gfCNCPoint4[2434] = {X 524.9094, Y 36.3306, Z -5.5000, A 0.000, B 0.000, C 0.000 }
gfCNCPoint4[2435] = {X 523.9717, Y 36.0380, Z -5.5000, A 0.000, B 0.000, C 0.000 }
gfCNCPoint4[2436] = {X 523.1116, Y 35.5636, Z -5.5000, A 0.000, B 0.000, C 0.000 }
gfCNCPoint4[2437] = {X 522.3639, Y 34.9265, Z -5.5000, A 0.000, B 0.000, C 0.000 }
gfCNCPoint4[2438] = {X 521.7590, Y 34.1525, Z -5.5000, A 0.000, B 0.000, C 0.000 }
gfCNCPoint4[2439] = {X 521.3213, Y 33.2731, Z -5.5000, A 0.000, B 0.000, C 0.000 }
gfCNCPoint4[2440] = {X 521.0686, Y 32.3239, Z -5.5000, A 0.000, B 0.000, C 0.000 }
gfCNCPoint4[2441] = {X 521.0222, Y 31.9379, Z -5.5000, A 0.000, B 0.000, C 0.000 }
gfCNCPoint4[2442] = {X 521.0068, Y 31.5494, Z -5.5000, A 0.000, B 0.000, C 0.000 }
gfCNCPoint4[2443] = {X 521.0076, Y 24.4815, Z -5.5000, A 0.000, B 0.000, C 0.000 }
gfCNCPoint4[2444] = {X 521.0984, Y 23.6300, Z -5.5000, A 0.000, B 0.000, C 0.000 }
gfCNCPoint4[2445] = {X 521.3368, Y 22.8074, Z -5.5000, A 0.000, B 0.000, C 0.000 }
gfCNCPoint4[2446] = {X 521.7152, Y 22.0391, Z -5.5000, A 0.000, B 0.000, C 0.000 }
gfCNCPoint4[2447] = {X 521.1864, Y 22.1316, Z -5.5000, A 0.000, B 0.000, C 0.000 }
gfCNCPoint4[2448] = {X 520.6505, Y 22.1656, Z -5.5000, A 0.000, B 0.000, C 0.000 }
gfCNCPoint4[2449] = {X 519.9691, Y 22.1657, Z -5.5000, A 0.000, B 0.000, C 0.000 }
gfCNCPoint4[2450] = {X 519.5109, Y 22.1442, Z -5.5000, A 0.000, B 0.000, C 0.000 }
gfCNCPoint4[2451] = {X 519.0567, Y 22.0797, Z -5.5000, A 0.000, B 0.000, C 0.000 }
gfCNCPoint4[2452] = {X 518.1336, Y 21.8074, Z -5.5000, A 0.000, B 0.000, C 0.000 }
gfCNCPoint4[2453] = {X 517.2820, Y 21.3592, Z -5.5000, A 0.000, B 0.000, C 0.000 }
gfCNCPoint4[2454] = {X 516.5348, Y 20.7527, Z -5.5000, A 0.000, B 0.000, C 0.000 }
gfCNCPoint4[2455] = {X 515.9212, Y 20.0113, Z -5.5000, A 0.000, B 0.000, C 0.000 }
gfCNCPoint4[2456] = {X 515.4650, Y 19.1639, Z -5.5000, A 0.000, B 0.000, C 0.000 }
gfCNCPoint4[2457] = {X 515.1840, Y 18.2434, Z -5.5000, A 0.000, B 0.000, C 0.000 }
gfCNCPoint4[2458] = {X 515.0891, Y 17.2857, Z -5.5000, A 0.000, B 0.000, C 0.000 }
gfCNCPoint4[2459] = {X 515.0891, Y 10.3077, Z -5.5000, A 0.000, B 0.000, C 0.000 }
gfCNCPoint4[2460] = {X 515.0966, Y 10.0382, Z -5.5000, A 0.000, B 0.000, C 0.000 }
gfCNCPoint4[2461] = {X 515.1189, Y 9.7696, Z -5.5000, A 0.000, B 0.000, C 0.000 }
gfCNCPoint4[2462] = {X 515.3252, Y 8.8083, Z -5.5000, A 0.000, B 0.000, C 0.000 }
gfCNCPoint4[2463] = {X 515.7199, Y 7.9079, Z -5.5000, A 0.000, B 0.000, C 0.000 }
gfCNCPoint4[2464] = {X 516.2872, Y 7.1049, Z -5.5000, A 0.000, B 0.000, C 0.000 }
gfCNCPoint4[2465] = {X 516.6493, Y 7.4200, Z -5.5000, A 0.000, B 0.000, C 0.000 }
gfCNCPoint4[2466] = {X 517.3374, Y 6.7815, Z -5.5000, A 0.000, B 0.000, C 0.000 }
gfCNCPoint4[2467] = {X 518.1451, Y 6.3035, Z -5.5000, A 0.000, B 0.000, C 0.000 }
gfCNCPoint4[2468] = {X 519.0359, Y 6.0078, Z -5.5000, A 0.000, B 0.000, C 0.000 }
gfCNCPoint4[2469] = {X 519.9692, Y 5.9077, Z -5.5000, A 0.000, B 0.000, C 0.000 }
gfCNCPoint4[2470] = {X 520.6509, Y 5.9079, Z -5.5000, A 0.000, B 0.000, C 0.000 }
gfCNCPoint4[2471] = {X 521.4832, Y 5.9951, Z -5.5000, A 0.000, B 0.000, C 0.000 }
gfCNCPoint4[2472] = {X 522.2840, Y 6.2382, Z -5.5000, A 0.000, B 0.000, C 0.000 }
gfCNCPoint4[2473] = {X 523.0242, Y 6.6287, Z -5.5000, A 0.000, B 0.000, C 0.000 }
gfCNCPoint4[2474] = {X 523.6771, Y 7.1522, Z -5.5000, A 0.000, B 0.000, C 0.000 }
gfCNCPoint4[2475] = {X 524.2191, Y 7.7898, Z -5.5000, A 0.000, B 0.000, C 0.000 }
gfCNCPoint4[2476] = {X 543.7489, Y 7.7902, Z -5.5000, A 0.000, B 0.000, C 0.000 }
gfCNCPoint4[2477] = {X 544.7471, Y 7.8776, Z -5.5000, A 0.000, B 0.000, C 0.000 }
gfCNCPoint4[2478] = {X 545.6998, Y 8.1882, Z -5.5000, A 0.000, B 0.000, C 0.000 }
gfCNCPoint4[2479] = {X 546.5576, Y 8.7062, Z -5.5000, A 0.000, B 0.000, C 0.000 }
gfCNCPoint4[2480] = {X 547.2761, Y 9.4046, Z -5.5000, A 0.000, B 0.000, C 0.000 }
gfCNCPoint4[2481] = {X 547.8182, Y 10.2474, Z -5.5000, A 0.000, B 0.000, C 0.000 }
gfCNCPoint4[2482] = {X 548.1558, Y 11.1908, Z -5.5000, A 0.000, B 0.000, C 0.000 }
gfCNCPoint4[2483] = {X 548.2714, Y 12.1862, Z -5.5000, A 0.000, B 0.000, C 0.000 }
gfCNCPoint4[2484] = {X 548.2712, Y 13.0233, Z -5.5000, A 0.000, B 0.000, C 0.000 }
gfCNCPoint4[2485] = {X 548.1630, Y 13.9487, Z -5.5000, A 0.000, B 0.000, C 0.000 }
gfCNCPoint4[2486] = {X 547.8624, Y 14.8306, Z -5.5000, A 0.000, B 0.000, C 0.000 }
gfCNCPoint4[2487] = {X 547.3828, Y 15.6295, Z -5.5000, A 0.000, B 0.000, C 0.000 }
gfCNCPoint4[2488] = {X 546.7458, Y 16.3094, Z -5.5000, A 0.000, B 0.000, C 0.000 }
gfCNCPoint4[2489] = {X 546.7444, Y 40.8762, Z -5.5000, A 0.000, B 0.000, C 0.000 }
gfCNCPoint4[2490] = {X 547.3888, Y 41.5653, Z -5.5000, A 0.000, B 0.000, C 0.000 }
gfCNCPoint4[2491] = {X 547.8715, Y 42.3759, Z -5.5000, A 0.000, B 0.000, C 0.000 }
gfCNCPoint4[2492] = {X 548.1703, Y 43.2708, Z -5.5000, A 0.000, B 0.000, C 0.000 }
gfCNCPoint4[2493] = {X 548.2714, Y 44.2089, Z -5.5000, A 0.000, B 0.000, C 0.000 }
gfCNCPoint4[2494] = {X 548.2714, Y 45.0006, Z -5.5000, A 0.000, B 0.000, C 0.000 }
gfCNCPoint4[2495] = {X 548.1558, Y 45.9960, Z -5.5000, A 0.000, B 0.000, C 0.000 }
gfCNCPoint4[2496] = {X 547.8182, Y 46.9394, Z -5.5000, A 0.000, B 0.000, C 0.000 }
gfCNCPoint4[2497] = {X 547.2761, Y 47.7821, Z -5.5000, A 0.000, B 0.000, C 0.000 }
gfCNCPoint4[2498] = {X 546.5576, Y 48.4805, Z -5.5000, A 0.000, B 0.000, C 0.000 }
gfCNCPoint4[2499] = {X 545.6998, Y 48.9984, Z -5.5000, A 0.000, B 0.000, C 0.000 }
gfCNCPoint4[2500] = {X 544.7471, Y 49.3090, Z -5.5000, A 0.000, B 0.000, C 0.000 }
gfCNCPoint4[2501] = {X 543.7489, Y 49.3963, Z -5.5000, A 0.000, B 0.000, C 0.000 }
gfCNCPoint4[2502] = {X 524.0863, Y 49.3967, Z -5.5000, A 0.000, B 0.000, C 0.000 }
gfCNCPoint4[2503] = {X 523.5296, Y 50.0317, Z -5.5000, A 0.000, B 0.000, C 0.000 }
gfCNCPoint4[2504] = {X 522.8651, Y 50.5530, Z -5.5000, A 0.000, B 0.000, C 0.000 }
gfCNCPoint4[2505] = {X 522.1159, Y 50.9428, Z -5.5000, A 0.000, B 0.000, C 0.000 }
gfCNCPoint4[2506] = {X 521.3077, Y 51.1876, Z -5.5000, A 0.000, B 0.000, C 0.000 }
gfCNCPoint4[2507] = {X 520.4681, Y 51.2791, Z -5.5000, A 0.000, B 0.000, C 0.000 }
gfCNCPoint4[2508] = {X 519.7998, Y 51.2791, Z -5.5000, A 0.000, B 0.000, C 0.000 }
gfCNCPoint4[2509] = {X 518.8207, Y 51.1688, Z -5.5000, A 0.000, B 0.000, C 0.000 }
gfCNCPoint4[2510] = {X 517.8907, Y 50.8434, Z -5.5000, A 0.000, B 0.000, C 0.000 }
gfCNCPoint4[2511] = {X 517.0564, Y 50.3192, Z -5.5000, A 0.000, B 0.000, C 0.000 }
gfCNCPoint4[2512] = {X 516.3597, Y 49.6225, Z -5.5000, A 0.000, B 0.000, C 0.000 }
gfCNCPoint4[2513] = {X 515.8355, Y 48.7882, Z -5.5000, A 0.000, B 0.000, C 0.000 }
gfCNCPoint4[2514] = {X 515.5101, Y 47.8582, Z -5.5000, A 0.000, B 0.000, C 0.000 }
gfCNCPoint4[2515] = {X 515.3998, Y 46.8791, Z -5.5000, A 0.000, B 0.000, C 0.000 }
gfCNCPoint4[2516] = {X 515.3998, Y 39.9011, Z -5.5000, A 0.000, B 0.000, C 0.000 }
gfCNCPoint4[2517] = {X 515.5101, Y 38.9220, Z -5.5000, A 0.000, B 0.000, C 0.000 }
gfCNCPoint4[2518] = {X 515.8355, Y 37.9920, Z -5.5000, A 0.000, B 0.000, C 0.000 }
gfCNCPoint4[2519] = {X 516.3597, Y 37.1577, Z -5.5000, A 0.000, B 0.000, C 0.000 }
gfCNCPoint4[2520] = {X 517.0564, Y 36.4610, Z -5.5000, A 0.000, B 0.000, C 0.000 }
gfCNCPoint4[2521] = {X 517.8907, Y 35.9368, Z -5.5000, A 0.000, B 0.000, C 0.000 }
gfCNCPoint4[2522] = {X 518.8207, Y 35.6114, Z -5.5000, A 0.000, B 0.000, C 0.000 }
gfCNCPoint4[2523] = {X 519.7998, Y 35.5011, Z -5.5000, A 0.000, B 0.000, C 0.000 }
gfCNCPoint4[2524] = {X 520.5280, Y 35.5015, Z -5.5000, A 0.000, B 0.000, C 0.000 }
gfCNCPoint4[2525] = {X 521.3613, Y 35.5927, Z -5.5000, A 0.000, B 0.000, C 0.000 }
gfCNCPoint4[2526] = {X 522.1622, Y 35.8403, Z -5.5000, A 0.000, B 0.000, C 0.000 }
gfCNCPoint4[2527] = {X 522.9017, Y 36.2353, Z -5.5000, A 0.000, B 0.000, C 0.000 }
gfCNCPoint4[2528] = {X 523.5527, Y 36.7633, Z -5.5000, A 0.000, B 0.000, C 0.000 }
gfCNCPoint4[2529] = {X 524.0919, Y 37.4053, Z -5.5000, A 0.000, B 0.000, C 0.000 }
gfCNCPoint4[2530] = {X 534.5519, Y 37.4057, Z -5.5000, A 0.000, B 0.000, C 0.000 }
gfCNCPoint4[2531] = {X 534.5519, Y 34.0457, Z -5.5000, A 0.000, B 0.000, C 0.000 }
gfCNCPoint4[2532] = {X 530.1520, Y 34.0454, Z -5.5000, A 0.000, B 0.000, C 0.000 }
gfCNCPoint4[2533] = {X 529.6043, Y 34.6957, Z -5.5000, A 0.000, B 0.000, C 0.000 }
gfCNCPoint4[2534] = {X 528.9418, Y 35.2285, Z -5.5000, A 0.000, B 0.000, C 0.000 }
gfCNCPoint4[2535] = {X 528.1892, Y 35.6240, Z -5.5000, A 0.000, B 0.000, C 0.000 }
gfCNCPoint4[2536] = {X 527.3745, Y 35.8673, Z -5.5000, A 0.000, B 0.000, C 0.000 }
gfCNCPoint4[2537] = {X 526.5283, Y 35.9495, Z -5.5000, A 0.000, B 0.000, C 0.000 }
gfCNCPoint4[2538] = {X 525.8868, Y 35.9495, Z -5.5000, A 0.000, B 0.000, C 0.000 }
gfCNCPoint4[2539] = {X 524.9077, Y 35.8391, Z -5.5000, A 0.000, B 0.000, C 0.000 }
gfCNCPoint4[2540] = {X 523.9777, Y 35.5137, Z -5.5000, A 0.000, B 0.000, C 0.000 }
gfCNCPoint4[2541] = {X 523.1434, Y 34.9895, Z -5.5000, A 0.000, B 0.000, C 0.000 }
gfCNCPoint4[2542] = {X 522.4467, Y 34.2928, Z -5.5000, A 0.000, B 0.000, C 0.000 }
gfCNCPoint4[2543] = {X 521.9225, Y 33.4585, Z -5.5000, A 0.000, B 0.000, C 0.000 }
gfCNCPoint4[2544] = {X 521.5971, Y 32.5285, Z -5.5000, A 0.000, B 0.000, C 0.000 }
gfCNCPoint4[2545] = {X 521.4868, Y 31.5495, Z -5.5000, A 0.000, B 0.000, C 0.000 }
gfCNCPoint4[2546] = {X 521.4868, Y 24.5714, Z -5.5000, A 0.000, B 0.000, C 0.000 }
gfCNCPoint4[2547] = {X 521.5971, Y 23.5923, Z -5.5000, A 0.000, B 0.000, C 0.000 }
gfCNCPoint4[2548] = {X 521.9225, Y 22.6623, Z -5.5000, A 0.000, B 0.000, C 0.000 }
gfCNCPoint4[2549] = {X 522.4467, Y 21.8281, Z -5.5000, A 0.000, B 0.000, C 0.000 }
gfCNCPoint4[2550] = {X 523.1434, Y 21.1314, Z -5.5000, A 0.000, B 0.000, C 0.000 }
gfCNCPoint4[2551] = {X 523.9777, Y 20.6072, Z -5.5000, A 0.000, B 0.000, C 0.000 }
gfCNCPoint4[2552] = {X 524.9077, Y 20.2817, Z -5.5000, A 0.000, B 0.000, C 0.000 }
gfCNCPoint4[2553] = {X 525.8868, Y 20.1714, Z -5.5000, A 0.000, B 0.000, C 0.000 }
gfCNCPoint4[2554] = {X 526.5702, Y 20.1716, Z -5.5000, A 0.000, B 0.000, C 0.000 }
gfCNCPoint4[2555] = {X 527.2691, Y 20.2342, Z -5.5000, A 0.000, B 0.000, C 0.000 }
gfCNCPoint4[2556] = {X 527.9491, Y 20.4071, Z -5.5000, A 0.000, B 0.000, C 0.000 }
gfCNCPoint4[2557] = {X 528.5930, Y 20.6859, Z -5.5000, A 0.000, B 0.000, C 0.000 }
gfCNCPoint4[2558] = {X 528.8182, Y 20.2620, Z -5.5000, A 0.000, B 0.000, C 0.000 }
gfCNCPoint4[2559] = {X 534.0719, Y 20.2621, Z -5.5000, A 0.000, B 0.000, C 0.000 }
gfCNCPoint4[2560] = {X 534.0719, Y 21.5737, Z -5.5000, A 0.000, B 0.000, C 0.000 }
gfCNCPoint4[2561] = {X 530.3790, Y 21.5735, Z -5.5000, A 0.000, B 0.000, C 0.000 }
gfCNCPoint4[2562] = {X 529.6679, Y 20.8353, Z -5.5000, A 0.000, B 0.000, C 0.000 }
gfCNCPoint4[2563] = {X 528.8182, Y 20.2620, Z -5.5000, A 0.000, B 0.000, C 0.000 }
gfCNCPoint4[2564] = {X 528.5930, Y 20.6859, Z -5.5000, A 0.000, B 0.000, C 0.000 }
gfCNCPoint4[2565] = {X 529.1776, Y 21.0584, Z -5.5000, A 0.000, B 0.000, C 0.000 }
gfCNCPoint4[2566] = {X 529.6965, Y 21.5180, Z -5.5000, A 0.000, B 0.000, C 0.000 }
gfCNCPoint4[2567] = {X 530.1368, Y 22.0535, Z -5.5000, A 0.000, B 0.000, C 0.000 }
gfCNCPoint4[2568] = {X 534.5519, Y 22.0537, Z -5.5000, A 0.000, B 0.000, C 0.000 }
gfCNCPoint4[2569] = {X 534.5519, Y 19.7821, Z -5.5000, A 0.000, B 0.000, C 0.000 }
gfCNCPoint4[2570] = {X 524.2342, Y 19.7819, Z -5.5000, A 0.000, B 0.000, C 0.000 }
gfCNCPoint4[2571] = {X 523.6865, Y 20.4321, Z -5.5000, A 0.000, B 0.000, C 0.000 }
gfCNCPoint4[2572] = {X 523.0240, Y 20.9649, Z -5.5000, A 0.000, B 0.000, C 0.000 }
gfCNCPoint4[2573] = {X 522.2715, Y 21.3603, Z -5.5000, A 0.000, B 0.000, C 0.000 }
gfCNCPoint4[2574] = {X 521.4569, Y 21.6036, Z -5.5000, A 0.000, B 0.000, C 0.000 }
gfCNCPoint4[2575] = {X 520.6107, Y 21.6857, Z -5.5000, A 0.000, B 0.000, C 0.000 }
gfCNCPoint4[2576] = {X 519.9691, Y 21.6857, Z -5.5000, A 0.000, B 0.000, C 0.000 }
gfCNCPoint4[2577] = {X 518.9900, Y 21.5754, Z -5.5000, A 0.000, B 0.000, C 0.000 }
gfCNCPoint4[2578] = {X 518.0600, Y 21.2500, Z -5.5000, A 0.000, B 0.000, C 0.000 }
gfCNCPoint4[2579] = {X 517.2257, Y 20.7258, Z -5.5000, A 0.000, B 0.000, C 0.000 }
gfCNCPoint4[2580] = {X 516.5290, Y 20.0291, Z -5.5000, A 0.000, B 0.000, C 0.000 }
gfCNCPoint4[2581] = {X 516.0048, Y 19.1948, Z -5.5000, A 0.000, B 0.000, C 0.000 }
gfCNCPoint4[2582] = {X 515.6794, Y 18.2648, Z -5.5000, A 0.000, B 0.000, C 0.000 }
gfCNCPoint4[2583] = {X 515.5691, Y 17.2857, Z -5.5000, A 0.000, B 0.000, C 0.000 }
gfCNCPoint4[2584] = {X 515.5691, Y 10.3077, Z -5.5000, A 0.000, B 0.000, C 0.000 }
gfCNCPoint4[2585] = {X 515.6394, Y 9.5244, Z -5.5000, A 0.000, B 0.000, C 0.000 }
gfCNCPoint4[2586] = {X 515.8480, Y 8.7661, Z -5.5000, A 0.000, B 0.000, C 0.000 }
gfCNCPoint4[2587] = {X 516.1883, Y 8.0571, Z -5.5000, A 0.000, B 0.000, C 0.000 }
gfCNCPoint4[2588] = {X 516.6493, Y 7.4200, Z -5.5000, A 0.000, B 0.000, C 0.000 }
gfCNCPoint4[2589] = {X 516.2872, Y 7.1049, Z -5.5000, A 0.000, B 0.000, C 0.000 }
gfCNCPoint4[2590] = {X 370.0950, Y 7.1049, Z -5.5000, A 0.000, B 0.000, C 0.000 }
gfCNCPoint4[2591] = {X 371.1183, Y 8.7931, Z -5.5000, A 0.000, B 0.000, C 0.000 }
gfCNCPoint4[2592] = {X 372.0301, Y 10.5439, Z -5.5000, A 0.000, B 0.000, C 0.000 }
gfCNCPoint4[2593] = {X 372.8770, Y 12.4761, Z -5.5000, A 0.000, B 0.000, C 0.000 }
gfCNCPoint4[2594] = {X 373.5881, Y 14.4624, Z -5.5000, A 0.000, B 0.000, C 0.000 }
gfCNCPoint4[2595] = {X 374.1600, Y 16.4931, Z -5.5000, A 0.000, B 0.000, C 0.000 }
gfCNCPoint4[2596] = {X 374.5900, Y 18.5585, Z -5.5000, A 0.000, B 0.000, C 0.000 }
gfCNCPoint4[2597] = {X 374.9577, Y 21.1545, Z -5.5000, A 0.000, B 0.000, C 0.000 }
gfCNCPoint4[2598] = {X 375.1412, Y 23.7700, Z -5.5000, A 0.000, B 0.000, C 0.000 }
gfCNCPoint4[2599] = {X 375.1394, Y 26.3919, Z -5.5000, A 0.000, B 0.000, C 0.000 }
gfCNCPoint4[2600] = {X 374.9524, Y 29.0072, Z -5.5000, A 0.000, B 0.000, C 0.000 }
gfCNCPoint4[2601] = {X 374.5811, Y 31.6027, Z -5.5000, A 0.000, B 0.000, C 0.000 }
gfCNCPoint4[2602] = {X 374.5614, Y 31.7151, Z -5.5000, A 0.000, B 0.000, C 0.000 }
gfCNCPoint4[2603] = {X 374.5412, Y 31.8274, Z -5.5000, A 0.000, B 0.000, C 0.000 }
gfCNCPoint4[2604] = {X 386.3479, Y 33.9724, Z -5.5000, A 0.000, B 0.000, C 0.000 }
gfCNCPoint4[2605] = {X 386.1166, Y 35.1498, Z -5.5000, A 0.000, B 0.000, C 0.000 }
gfCNCPoint4[2606] = {X 385.8517, Y 36.3200, Z -5.5000, A 0.000, B 0.000, C 0.000 }
gfCNCPoint4[2607] = {X 386.9552, Y 36.3200, Z -5.5000, A 0.000, B 0.000, C 0.000 }
gfCNCPoint4[2608] = {X 386.9552, Y 35.0284, Z -5.5000, A 0.000, B 0.000, C 0.000 }
gfCNCPoint4[2609] = {X 386.3479, Y 33.9724, Z -5.5000, A 0.000, B 0.000, C 0.000 }
gfCNCPoint4[2610] = {X 383.9866, Y 33.5434, Z -5.5000, A 0.000, B 0.000, C 0.000 }
gfCNCPoint4[2611] = {X 383.7685, Y 34.6534, Z -5.5000, A 0.000, B 0.000, C 0.000 }
gfCNCPoint4[2612] = {X 383.5187, Y 35.7567, Z -5.5000, A 0.000, B 0.000, C 0.000 }
gfCNCPoint4[2613] = {X 383.1281, Y 37.2465, Z -5.5000, A 0.000, B 0.000, C 0.000 }
gfCNCPoint4[2614] = {X 382.6798, Y 38.7200, Z -5.5000, A 0.000, B 0.000, C 0.000 }
gfCNCPoint4[2615] = {X 388.0597, Y 38.7200, Z -5.5000, A 0.000, B 0.000, C 0.000 }
gfCNCPoint4[2616] = {X 388.4821, Y 38.7246, Z -5.5000, A 0.000, B 0.000, C 0.000 }
gfCNCPoint4[2617] = {X 388.9042, Y 38.7385, Z -5.5000, A 0.000, B 0.000, C 0.000 }
gfCNCPoint4[2618] = {X 389.1203, Y 38.2363, Z -5.5000, A 0.000, B 0.000, C 0.000 }
gfCNCPoint4[2619] = {X 389.3552, Y 37.7426, Z -5.5000, A 0.000, B 0.000, C 0.000 }
gfCNCPoint4[2620] = {X 389.3552, Y 34.3876, Z -5.5000, A 0.000, B 0.000, C 0.000 }
gfCNCPoint4[2621] = {X 384.7450, Y 26.3706, Z -5.5000, A 0.000, B 0.000, C 0.000 }
gfCNCPoint4[2622] = {X 384.6225, Y 28.6819, Z -5.5000, A 0.000, B 0.000, C 0.000 }
gfCNCPoint4[2623] = {X 384.3856, Y 30.9844, Z -5.5000, A 0.000, B 0.000, C 0.000 }
gfCNCPoint4[2624] = {X 384.0349, Y 33.2722, Z -5.5000, A 0.000, B 0.000, C 0.000 }
gfCNCPoint4[2625] = {X 384.0110, Y 33.4079, Z -5.5000, A 0.000, B 0.000, C 0.000 }
gfCNCPoint4[2626] = {X 383.9866, Y 33.5434, Z -5.5000, A 0.000, B 0.000, C 0.000 }
gfCNCPoint4[2627] = {X 381.6252, Y 33.1144, Z -5.5000, A 0.000, B 0.000, C 0.000 }
gfCNCPoint4[2628] = {X 381.0937, Y 35.5664, Z -5.5000, A 0.000, B 0.000, C 0.000 }
gfCNCPoint4[2629] = {X 380.3978, Y 37.9769, Z -5.5000, A 0.000, B 0.000, C 0.000 }
gfCNCPoint4[2630] = {X 379.8417, Y 39.5618, Z -5.5000, A 0.000, B 0.000, C 0.000 }
gfCNCPoint4[2631] = {X 379.2146, Y 41.1200, Z -5.5000, A 0.000, B 0.000, C 0.000 }
gfCNCPoint4[2632] = {X 388.0597, Y 41.1200, Z -5.5000, A 0.000, B 0.000, C 0.000 }
gfCNCPoint4[2633] = {X 389.3255, Y 41.1675, Z -5.5000, A 0.000, B 0.000, C 0.000 }
gfCNCPoint4[2634] = {X 390.5842, Y 41.3098, Z -5.5000, A 0.000, B 0.000, C 0.000 }
gfCNCPoint4[2635] = {X 391.0709, Y 39.7837, Z -5.5000, A 0.000, B 0.000, C 0.000 }
gfCNCPoint4[2636] = {X 391.7552, Y 38.3354, Z -5.5000, A 0.000, B 0.000, C 0.000 }
gfCNCPoint4[2637] = {X 391.7552, Y 33.7467, Z -5.5000, A 0.000, B 0.000, C 0.000 }
gfCNCPoint4[2638] = {X 386.7908, Y 25.1137, Z -5.5000, A 0.000, B 0.000, C 0.000 }
gfCNCPoint4[2639] = {X 386.1520, Y 24.0220, Z -5.5000, A 0.000, B 0.000, C 0.000 }
gfCNCPoint4[2640] = {X 385.4969, Y 22.9400, Z -5.5000, A 0.000, B 0.000, C 0.000 }
gfCNCPoint4[2641] = {X 384.4706, Y 22.1520, Z -5.5000, A 0.000, B 0.000, C 0.000 }
gfCNCPoint4[2642] = {X 383.5345, Y 21.2589, Z -5.5000, A 0.000, B 0.000, C 0.000 }
gfCNCPoint4[2643] = {X 382.6993, Y 20.2707, Z -5.5000, A 0.000, B 0.000, C 0.000 }
gfCNCPoint4[2644] = {X 381.9745, Y 19.1988, Z -5.5000, A 0.000, B 0.000, C 0.000 }
gfCNCPoint4[2645] = {X 382.2252, Y 21.5591, Z -5.5000, A 0.000, B 0.000, C 0.000 }
gfCNCPoint4[2646] = {X 382.3492, Y 23.9294, Z -5.5000, A 0.000, B 0.000, C 0.000 }
gfCNCPoint4[2647] = {X 382.3459, Y 26.3030, Z -5.5000, A 0.000, B 0.000, C 0.000 }
gfCNCPoint4[2648] = {X 382.2296, Y 28.4972, Z -5.5000, A 0.000, B 0.000, C 0.000 }
gfCNCPoint4[2649] = {X 382.0046, Y 30.6829, Z -5.5000, A 0.000, B 0.000, C 0.000 }
gfCNCPoint4[2650] = {X 381.6714, Y 32.8548, Z -5.5000, A 0.000, B 0.000, C 0.000 }
gfCNCPoint4[2651] = {X 381.6486, Y 32.9846, Z -5.5000, A 0.000, B 0.000, C 0.000 }
gfCNCPoint4[2652] = {X 381.6252, Y 33.1144, Z -5.5000, A 0.000, B 0.000, C 0.000 }
gfCNCPoint4[2653] = {X 379.2639, Y 32.6854, Z -5.5000, A 0.000, B 0.000, C 0.000 }
gfCNCPoint4[2654] = {X 378.7008, Y 35.2357, Z -5.5000, A 0.000, B 0.000, C 0.000 }
gfCNCPoint4[2655] = {X 377.9477, Y 37.7366, Z -5.5000, A 0.000, B 0.000, C 0.000 }
gfCNCPoint4[2656] = {X 377.0090, Y 40.1738, Z -5.5000, A 0.000, B 0.000, C 0.000 }
gfCNCPoint4[2657] = {X 376.2271, Y 41.8691, Z -5.5000, A 0.000, B 0.000, C 0.000 }
gfCNCPoint4[2658] = {X 375.3553, Y 43.5200, Z -5.5000, A 0.000, B 0.000, C 0.000 }
gfCNCPoint4[2659] = {X 388.0597, Y 43.5200, Z -5.5000, A 0.000, B 0.000, C 0.000 }
gfCNCPoint4[2660] = {X 389.6072, Y 43.6029, Z -5.5000, A 0.000, B 0.000, C 0.000 }
gfCNCPoint4[2661] = {X 391.1370, Y 43.8508, Z -5.5000, A 0.000, B 0.000, C 0.000 }
gfCNCPoint4[2662] = {X 392.6316, Y 44.2607, Z -5.5000, A 0.000, B 0.000, C 0.000 }
gfCNCPoint4[2663] = {X 392.6316, Y 44.1162, Z -5.5000, A 0.000, B 0.000, C 0.000 }
gfCNCPoint4[2664] = {X 392.7390, Y 42.7683, Z -5.5000, A 0.000, B 0.000, C 0.000 }
gfCNCPoint4[2665] = {X 393.0331, Y 41.4485, Z -5.5000, A 0.000, B 0.000, C 0.000 }
gfCNCPoint4[2666] = {X 393.5083, Y 40.1826, Z -5.5000, A 0.000, B 0.000, C 0.000 }
gfCNCPoint4[2667] = {X 394.1552, Y 38.9952, Z -5.5000, A 0.000, B 0.000, C 0.000 }
gfCNCPoint4[2668] = {X 394.1552, Y 33.1058, Z -5.5000, A 0.000, B 0.000, C 0.000 }
gfCNCPoint4[2669] = {X 388.8713, Y 23.9173, Z -5.5000, A 0.000, B 0.000, C 0.000 }
gfCNCPoint4[2670] = {X 388.0755, Y 22.5620, Z -5.5000, A 0.000, B 0.000, C 0.000 }
gfCNCPoint4[2671] = {X 387.2552, Y 21.2214, Z -5.5000, A 0.000, B 0.000, C 0.000 }
gfCNCPoint4[2672] = {X 386.3086, Y 20.5576, Z -5.5000, A 0.000, B 0.000, C 0.000 }
gfCNCPoint4[2673] = {X 385.4479, Y 19.7857, Z -5.5000, A 0.000, B 0.000, C 0.000 }
gfCNCPoint4[2674] = {X 384.6853, Y 18.9166, Z -5.5000, A 0.000, B 0.000, C 0.000 }
gfCNCPoint4[2675] = {X 384.0318, Y 17.9629, Z -5.5000, A 0.000, B 0.000, C 0.000 }
gfCNCPoint4[2676] = {X 383.4420, Y 16.8138, Z -5.5000, A 0.000, B 0.000, C 0.000 }
gfCNCPoint4[2677] = {X 383.0105, Y 15.5964, Z -5.5000, A 0.000, B 0.000, C 0.000 }
gfCNCPoint4[2678] = {X 382.7448, Y 14.3324, Z -5.5000, A 0.000, B 0.000, C 0.000 }
gfCNCPoint4[2679] = {X 382.6498, Y 13.0443, Z -5.5000, A 0.000, B 0.000, C 0.000 }
gfCNCPoint4[2680] = {X 382.6496, Y 12.1868, Z -5.5000, A 0.000, B 0.000, C 0.000 }
gfCNCPoint4[2681] = {X 382.6507, Y 12.0459, Z -5.5000, A 0.000, B 0.000, C 0.000 }
gfCNCPoint4[2682] = {X 382.6537, Y 11.9049, Z -5.5000, A 0.000, B 0.000, C 0.000 }
gfCNCPoint4[2683] = {X 377.7902, Y 11.9049, Z -5.5000, A 0.000, B 0.000, C 0.000 }
gfCNCPoint4[2684] = {X 378.4099, Y 13.8167, Z -5.5000, A 0.000, B 0.000, C 0.000 }
gfCNCPoint4[2685] = {X 378.9198, Y 15.7606, Z -5.5000, A 0.000, B 0.000, C 0.000 }
gfCNCPoint4[2686] = {X 379.3180, Y 17.7305, Z -5.5000, A 0.000, B 0.000, C 0.000 }
gfCNCPoint4[2687] = {X 379.4665, Y 18.6218, Z -5.5000, A 0.000, B 0.000, C 0.000 }
gfCNCPoint4[2688] = {X 379.5956, Y 19.5162, Z -5.5000, A 0.000, B 0.000, C 0.000 }
gfCNCPoint4[2689] = {X 379.8589, Y 22.0976, Z -5.5000, A 0.000, B 0.000, C 0.000 }
gfCNCPoint4[2690] = {X 379.9619, Y 24.6904, Z -5.5000, A 0.000, B 0.000, C 0.000 }
gfCNCPoint4[2691] = {X 379.9042, Y 27.2846, Z -5.5000, A 0.000, B 0.000, C 0.000 }
gfCNCPoint4[2692] = {X 379.6859, Y 29.8702, Z -5.5000, A 0.000, B 0.000, C 0.000 }
gfCNCPoint4[2693] = {X 379.3080, Y 32.4374, Z -5.5000, A 0.000, B 0.000, C 0.000 }
gfCNCPoint4[2694] = {X 379.2862, Y 32.5614, Z -5.5000, A 0.000, B 0.000, C 0.000 }
gfCNCPoint4[2695] = {X 379.2639, Y 32.6854, Z -5.5000, A 0.000, B 0.000, C 0.000 }
gfCNCPoint4[2696] = {X 376.9025, Y 32.2564, Z -5.5000, A 0.000, B 0.000, C 0.000 }
gfCNCPoint4[2697] = {X 376.3115, Y 34.8830, Z -5.5000, A 0.000, B 0.000, C 0.000 }
gfCNCPoint4[2698] = {X 375.5040, Y 37.4513, Z -5.5000, A 0.000, B 0.000, C 0.000 }
gfCNCPoint4[2699] = {X 374.4858, Y 39.9437, Z -5.5000, A 0.000, B 0.000, C 0.000 }
gfCNCPoint4[2700] = {X 373.2639, Y 42.3427, Z -5.5000, A 0.000, B 0.000, C 0.000 }
gfCNCPoint4[2701] = {X 372.1889, Y 44.1167, Z -5.5000, A 0.000, B 0.000, C 0.000 }
gfCNCPoint4[2702] = {X 371.0024, Y 45.8182, Z -5.5000, A 0.000, B 0.000, C 0.000 }
gfCNCPoint4[2703] = {X 370.9154, Y 45.9351, Z -5.5000, A 0.000, B 0.000, C 0.000 }
gfCNCPoint4[2704] = {X 371.2172, Y 45.9238, Z -5.5000, A 0.000, B 0.000, C 0.000 }
gfCNCPoint4[2705] = {X 371.5193, Y 45.9200, Z -5.5000, A 0.000, B 0.000, C 0.000 }
gfCNCPoint4[2706] = {X 388.0597, Y 45.9200, Z -5.5000, A 0.000, B 0.000, C 0.000 }
gfCNCPoint4[2707] = {X 389.4143, Y 45.9962, Z -5.5000, A 0.000, B 0.000, C 0.000 }
gfCNCPoint4[2708] = {X 390.7519, Y 46.2238, Z -5.5000, A 0.000, B 0.000, C 0.000 }
gfCNCPoint4[2709] = {X 392.0555, Y 46.6000, Z -5.5000, A 0.000, B 0.000, C 0.000 }
gfCNCPoint4[2710] = {X 393.3087, Y 47.1200, Z -5.5000, A 0.000, B 0.000, C 0.000 }
gfCNCPoint4[2711] = {X 394.2237, Y 46.7243, Z -5.5000, A 0.000, B 0.000, C 0.000 }
gfCNCPoint4[2712] = {X 395.1681, Y 46.4053, Z -5.5000, A 0.000, B 0.000, C 0.000 }
gfCNCPoint4[2713] = {X 395.0678, Y 45.7292, Z -5.5000, A 0.000, B 0.000, C 0.000 }
gfCNCPoint4[2714] = {X 395.0314, Y 45.0468, Z -5.5000, A 0.000, B 0.000, C 0.000 }
gfCNCPoint4[2715] = {X 395.0316, Y 44.1297, Z -5.5000, A 0.000, B 0.000, C 0.000 }
gfCNCPoint4[2716] = {X 395.1397, Y 42.9565, Z -5.5000, A 0.000, B 0.000, C 0.000 }
gfCNCPoint4[2717] = {X 395.4356, Y 41.8161, Z -5.5000, A 0.000, B 0.000, C 0.000 }
gfCNCPoint4[2718] = {X 395.9116, Y 40.7384, Z -5.5000, A 0.000, B 0.000, C 0.000 }
gfCNCPoint4[2719] = {X 396.5552, Y 39.7516, Z -5.5000, A 0.000, B 0.000, C 0.000 }
gfCNCPoint4[2720] = {X 396.5552, Y 32.4650, Z -5.5000, A 0.000, B 0.000, C 0.000 }
gfCNCPoint4[2721] = {X 390.9518, Y 22.7209, Z -5.5000, A 0.000, B 0.000, C 0.000 }
gfCNCPoint4[2722] = {X 390.0923, Y 21.2587, Z -5.5000, A 0.000, B 0.000, C 0.000 }
gfCNCPoint4[2723] = {X 389.2052, Y 19.8131, Z -5.5000, A 0.000, B 0.000, C 0.000 }
gfCNCPoint4[2724] = {X 389.0620, Y 19.6021, Z -5.5000, A 0.000, B 0.000, C 0.000 }
gfCNCPoint4[2725] = {X 388.9042, Y 19.4018, Z -5.5000, A 0.000, B 0.000, C 0.000 }
gfCNCPoint4[2726] = {X 387.8160, Y 18.6899, Z -5.5000, A 0.000, B 0.000, C 0.000 }
gfCNCPoint4[2727] = {X 386.8719, Y 17.7958, Z -5.5000, A 0.000, B 0.000, C 0.000 }
gfCNCPoint4[2728] = {X 386.1018, Y 16.7480, Z -5.5000, A 0.000, B 0.000, C 0.000 }
gfCNCPoint4[2729] = {X 385.5305, Y 15.5799, Z -5.5000, A 0.000, B 0.000, C 0.000 }
gfCNCPoint4[2730] = {X 385.1760, Y 14.3288, Z -5.5000, A 0.000, B 0.000, C 0.000 }
gfCNCPoint4[2731] = {X 385.0498, Y 13.0347, Z -5.5000, A 0.000, B 0.000, C 0.000 }
gfCNCPoint4[2732] = {X 385.0496, Y 12.1868, Z -5.5000, A 0.000, B 0.000, C 0.000 }
gfCNCPoint4[2733] = {X 385.0504, Y 12.0808, Z -5.5000, A 0.000, B 0.000, C 0.000 }
gfCNCPoint4[2734] = {X 385.0527, Y 11.9748, Z -5.5000, A 0.000, B 0.000, C 0.000 }
gfCNCPoint4[2735] = {X 385.1994, Y 10.7177, Z -5.5000, A 0.000, B 0.000, C 0.000 }
gfCNCPoint4[2736] = {X 385.5616, Y 9.5049, Z -5.5000, A 0.000, B 0.000, C 0.000 }
gfCNCPoint4[2737] = {X 374.1936, Y 9.5049, Z -5.5000, A 0.000, B 0.000, C 0.000 }
gfCNCPoint4[2738] = {X 374.9037, Y 11.0897, Z -5.5000, A 0.000, B 0.000, C 0.000 }
gfCNCPoint4[2739] = {X 375.5292, Y 12.7098, Z -5.5000, A 0.000, B 0.000, C 0.000 }
gfCNCPoint4[2740] = {X 376.1073, Y 14.4933, Z -5.5000, A 0.000, B 0.000, C 0.000 }
gfCNCPoint4[2741] = {X 376.5828, Y 16.3068, Z -5.5000, A 0.000, B 0.000, C 0.000 }
gfCNCPoint4[2742] = {X 376.9540, Y 18.1445, Z -5.5000, A 0.000, B 0.000, C 0.000 }
gfCNCPoint4[2743] = {X 377.3449, Y 20.9060, Z -5.5000, A 0.000, B 0.000, C 0.000 }
gfCNCPoint4[2744] = {X 377.5398, Y 23.6882, Z -5.5000, A 0.000, B 0.000, C 0.000 }
gfCNCPoint4[2745] = {X 377.5379, Y 26.4772, Z -5.5000, A 0.000, B 0.000, C 0.000 }
gfCNCPoint4[2746] = {X 377.3392, Y 29.2591, Z -5.5000, A 0.000, B 0.000, C 0.000 }
gfCNCPoint4[2747] = {X 376.9446, Y 32.0200, Z -5.5000, A 0.000, B 0.000, C 0.000 }
gfCNCPoint4[2748] = {X 376.9238, Y 32.1382, Z -5.5000, A 0.000, B 0.000, C 0.000 }
gfCNCPoint4[2749] = {X 376.9025, Y 32.2564, Z -5.5000, A 0.000, B 0.000, C 0.000 }
gfCNCPoint4[2750] = {X 374.5412, Y 31.8274, Z -5.5000, A 0.000, B 0.000, C 0.000 }
gfCNCPoint4[2751] = {X 374.0428, Y 34.0754, Z -5.5000, A 0.000, B 0.000, C 0.000 }
gfCNCPoint4[2752] = {X 373.3732, Y 36.2784, Z -5.5000, A 0.000, B 0.000, C 0.000 }
gfCNCPoint4[2753] = {X 372.5363, Y 38.4235, Z -5.5000, A 0.000, B 0.000, C 0.000 }
gfCNCPoint4[2754] = {X 371.5371, Y 40.4979, Z -5.5000, A 0.000, B 0.000, C 0.000 }
gfCNCPoint4[2755] = {X 370.3815, Y 42.4895, Z -5.5000, A 0.000, B 0.000, C 0.000 }
gfCNCPoint4[2756] = {X 369.0763, Y 44.3864, Z -5.5000, A 0.000, B 0.000, C 0.000 }
gfCNCPoint4[2757] = {X 369.0351, Y 44.4418, Z -5.5000, A 0.000, B 0.000, C 0.000 }
gfCNCPoint4[2758] = {X 368.9938, Y 44.4972, Z -5.5000, A 0.000, B 0.000, C 0.000 }
gfCNCPoint4[2759] = {X 367.5945, Y 46.2171, Z -5.5000, A 0.000, B 0.000, C 0.000 }
gfCNCPoint4[2760] = {X 366.0605, Y 47.8180, Z -5.5000, A 0.000, B 0.000, C 0.000 }
gfCNCPoint4[2761] = {X 364.4019, Y 49.2893, Z -5.5000, A 0.000, B 0.000, C 0.000 }
gfCNCPoint4[2762] = {X 362.6295, Y 50.6214, Z -5.5000, A 0.000, B 0.000, C 0.000 }
gfCNCPoint4[2763] = {X 360.7550, Y 51.8056, Z -5.5000, A 0.000, B 0.000, C 0.000 }
gfCNCPoint4[2764] = {X 358.7907, Y 52.8340, Z -5.5000, A 0.000, B 0.000, C 0.000 }
gfCNCPoint4[2765] = {X 358.6059, Y 52.9205, Z -5.5000, A 0.000, B 0.000, C 0.000 }
gfCNCPoint4[2766] = {X 358.4204, Y 53.0057, Z -5.5000, A 0.000, B 0.000, C 0.000 }
gfCNCPoint4[2767] = {X 356.1469, Y 53.8824, Z -5.5000, A 0.000, B 0.000, C 0.000 }
gfCNCPoint4[2768] = {X 353.8066, Y 54.5609, Z -5.5000, A 0.000, B 0.000, C 0.000 }
gfCNCPoint4[2769] = {X 351.4167, Y 55.0361, Z -5.5000, A 0.000, B 0.000, C 0.000 }
gfCNCPoint4[2770] = {X 348.9948, Y 55.3046, Z -5.5000, A 0.000, B 0.000, C 0.000 }
gfCNCPoint4[2771] = {X 349.9659, Y 69.6719, Z -5.5000, A 0.000, B 0.000, C 0.000 }
gfCNCPoint4[2772] = {X 348.6647, Y 69.7399, Z -5.5000, A 0.000, B 0.000, C 0.000 }
gfCNCPoint4[2773] = {X 347.3621, Y 69.7683, Z -5.5000, A 0.000, B 0.000, C 0.000 }
gfCNCPoint4[2774] = {X 346.5844, Y 69.7775, Z -5.5000, A 0.000, B 0.000, C 0.000 }
gfCNCPoint4[2775] = {X 345.8068, Y 69.7727, Z -5.5000, A 0.000, B 0.000, C 0.000 }
gfCNCPoint4[2776] = {X 345.5910, Y 70.1904, Z -5.5000, A 0.000, B 0.000, C 0.000 }
gfCNCPoint4[2777] = {X 345.3671, Y 70.6038, Z -5.5000, A 0.000, B 0.000, C 0.000 }
gfCNCPoint4[2778] = {X 347.2075, Y 70.6211, Z -5.5000, A 0.000, B 0.000, C 0.000 }
gfCNCPoint4[2779] = {X 349.0480, Y 70.6094, Z -5.5000, A 0.000, B 0.000, C 0.000 }
gfCNCPoint4[2780] = {X 349.7519, Y 70.6091, Z -5.5000, A 0.000, B 0.000, C 0.000 }
gfCNCPoint4[2781] = {X 350.4558, Y 70.6035, Z -5.5000, A 0.000, B 0.000, C 0.000 }
gfCNCPoint4[2782] = {X 350.2058, Y 70.1404, Z -5.5000, A 0.000, B 0.000, C 0.000 }
gfCNCPoint4[2783] = {X 349.9659, Y 69.6719, Z -5.5000, A 0.000, B 0.000, C 0.000 }
gfCNCPoint4[2784] = {X 349.8041, Y 67.2773, Z -5.5000, A 0.000, B 0.000, C 0.000 }
gfCNCPoint4[2785] = {X 348.5674, Y 67.3419, Z -5.5000, A 0.000, B 0.000, C 0.000 }
gfCNCPoint4[2786] = {X 347.3294, Y 67.3685, Z -5.5000, A 0.000, B 0.000, C 0.000 }
gfCNCPoint4[2787] = {X 345.8126, Y 67.3725, Z -5.5000, A 0.000, B 0.000, C 0.000 }
gfCNCPoint4[2788] = {X 344.2967, Y 67.3207, Z -5.5000, A 0.000, B 0.000, C 0.000 }
gfCNCPoint4[2789] = {X 343.8111, Y 68.3945, Z -5.5000, A 0.000, B 0.000, C 0.000 }
gfCNCPoint4[2790] = {X 343.2680, Y 69.4403, Z -5.5000, A 0.000, B 0.000, C 0.000 }
gfCNCPoint4[2791] = {X 342.7880, Y 70.2631, Z -5.5000, A 0.000, B 0.000, C 0.000 }
gfCNCPoint4[2792] = {X 342.2725, Y 71.0640, Z -5.5000, A 0.000, B 0.000, C 0.000 }
gfCNCPoint4[2793] = {X 342.2727, Y 72.9114, Z -5.5000, A 0.000, B 0.000, C 0.000 }
gfCNCPoint4[2794] = {X 343.7988, Y 72.9672, Z -5.5000, A 0.000, B 0.000, C 0.000 }
gfCNCPoint4[2795] = {X 345.3256, Y 73.0034, Z -5.5000, A 0.000, B 0.000, C 0.000 }
gfCNCPoint4[2796] = {X 347.1933, Y 73.0211, Z -5.5000, A 0.000, B 0.000, C 0.000 }
gfCNCPoint4[2797] = {X 349.0612, Y 73.0095, Z -5.5000, A 0.000, B 0.000, C 0.000 }
gfCNCPoint4[2798] = {X 349.7724, Y 73.0090, Z -5.5000, A 0.000, B 0.000, C 0.000 }
gfCNCPoint4[2799] = {X 350.4837, Y 73.0034, Z -5.5000, A 0.000, B 0.000, C 0.000 }
gfCNCPoint4[2800] = {X 352.0217, Y 72.9733, Z -5.5000, A 0.000, B 0.000, C 0.000 }
gfCNCPoint4[2801] = {X 353.5590, Y 72.9188, Z -5.5000, A 0.000, B 0.000, C 0.000 }
gfCNCPoint4[2802] = {X 353.5589, Y 71.0769, Z -5.5000, A 0.000, B 0.000, C 0.000 }
gfCNCPoint4[2803] = {X 353.0389, Y 70.2698, Z -5.5000, A 0.000, B 0.000, C 0.000 }
gfCNCPoint4[2804] = {X 352.5551, Y 69.4405, Z -5.5000, A 0.000, B 0.000, C 0.000 }
gfCNCPoint4[2805] = {X 351.9680, Y 68.3027, Z -5.5000, A 0.000, B 0.000, C 0.000 }
gfCNCPoint4[2806] = {X 351.4491, Y 67.1323, Z -5.5000, A 0.000, B 0.000, C 0.000 }
gfCNCPoint4[2807] = {X 350.6273, Y 67.2132, Z -5.5000, A 0.000, B 0.000, C 0.000 }
gfCNCPoint4[2808] = {X 349.8041, Y 67.2773, Z -5.5000, A 0.000, B 0.000, C 0.000 }
gfCNCPoint4[2809] = {X 349.6422, Y 64.8828, Z -5.5000, A 0.000, B 0.000, C 0.000 }
gfCNCPoint4[2810] = {X 348.4701, Y 64.9438, Z -5.5000, A 0.000, B 0.000, C 0.000 }
gfCNCPoint4[2811] = {X 347.2967, Y 64.9686, Z -5.5000, A 0.000, B 0.000, C 0.000 }
gfCNCPoint4[2812] = {X 344.9827, Y 64.9495, Z -5.5000, A 0.000, B 0.000, C 0.000 }
gfCNCPoint4[2813] = {X 342.6739, Y 64.7922, Z -5.5000, A 0.000, B 0.000, C 0.000 }
gfCNCPoint4[2814] = {X 341.9393, Y 66.7269, Z -5.5000, A 0.000, B 0.000, C 0.000 }
gfCNCPoint4[2815] = {X 341.0018, Y 68.5720, Z -5.5000, A 0.000, B 0.000, C 0.000 }
gfCNCPoint4[2816] = {X 339.8724, Y 70.3061, Z -5.5000, A 0.000, B 0.000, C 0.000 }
gfCNCPoint4[2817] = {X 339.8729, Y 75.1887, Z -5.5000, A 0.000, B 0.000, C 0.000 }
gfCNCPoint4[2818] = {X 344.4716, Y 75.3863, Z -5.5000, A 0.000, B 0.000, C 0.000 }
gfCNCPoint4[2819] = {X 349.0745, Y 75.4095, Z -5.5000, A 0.000, B 0.000, C 0.000 }
gfCNCPoint4[2820] = {X 352.5187, Y 75.3596, Z -5.5000, A 0.000, B 0.000, C 0.000 }
gfCNCPoint4[2821] = {X 355.9592, Y 75.1904, Z -5.5000, A 0.000, B 0.000, C 0.000 }
gfCNCPoint4[2822] = {X 355.9589, Y 70.3179, Z -5.5000, A 0.000, B 0.000, C 0.000 }
gfCNCPoint4[2823] = {X 355.0511, Y 68.9600, Z -5.5000, A 0.000, B 0.000, C 0.000 }
gfCNCPoint4[2824] = {X 354.2616, Y 67.5300, Z -5.5000, A 0.000, B 0.000, C 0.000 }
gfCNCPoint4[2825] = {X 353.5959, Y 66.0384, Z -5.5000, A 0.000, B 0.000, C 0.000 }
gfCNCPoint4[2826] = {X 353.0589, Y 64.4959, Z -5.5000, A 0.000, B 0.000, C 0.000 }
gfCNCPoint4[2827] = {X 351.3550, Y 64.7280, Z -5.5000, A 0.000, B 0.000, C 0.000 }
gfCNCPoint4[2828] = {X 349.6422, Y 64.8828, Z -5.5000, A 0.000, B 0.000, C 0.000 }
gfCNCPoint4[2829] = {X 349.4804, Y 62.4882, Z -5.5000, A 0.000, B 0.000, C 0.000 }
gfCNCPoint4[2830] = {X 348.3728, Y 62.5458, Z -5.5000, A 0.000, B 0.000, C 0.000 }
gfCNCPoint4[2831] = {X 347.2640, Y 62.5688, Z -5.5000, A 0.000, B 0.000, C 0.000 }
gfCNCPoint4[2832] = {X 345.1285, Y 62.5532, Z -5.5000, A 0.000, B 0.000, C 0.000 }
gfCNCPoint4[2833] = {X 342.9975, Y 62.4124, Z -5.5000, A 0.000, B 0.000, C 0.000 }
gfCNCPoint4[2834] = {X 340.8786, Y 62.1466, Z -5.5000, A 0.000, B 0.000, C 0.000 }
gfCNCPoint4[2835] = {X 340.4888, Y 63.7345, Z -5.5000, A 0.000, B 0.000, C 0.000 }
gfCNCPoint4[2836] = {X 339.9475, Y 65.2772, Z -5.5000, A 0.000, B 0.000, C 0.000 }
gfCNCPoint4[2837] = {X 339.2598, Y 66.7605, Z -5.5000, A 0.000, B 0.000, C 0.000 }
gfCNCPoint4[2838] = {X 338.4322, Y 68.1706, Z -5.5000, A 0.000, B 0.000, C 0.000 }
gfCNCPoint4[2839] = {X 337.4724, Y 69.4941, Z -5.5000, A 0.000, B 0.000, C 0.000 }
gfCNCPoint4[2840] = {X 337.4731, Y 77.4240, Z -5.5000, A 0.000, B 0.000, C 0.000 }
gfCNCPoint4[2841] = {X 341.3400, Y 77.6736, Z -5.5000, A 0.000, B 0.000, C 0.000 }
gfCNCPoint4[2842] = {X 345.2128, Y 77.8022, Z -5.5000, A 0.000, B 0.000, C 0.000 }
gfCNCPoint4[2843] = {X 349.0878, Y 77.8096, Z -5.5000, A 0.000, B 0.000, C 0.000 }
gfCNCPoint4[2844] = {X 353.7281, Y 77.7160, Z -5.5000, A 0.000, B 0.000, C 0.000 }
gfCNCPoint4[2845] = {X 358.3593, Y 77.4111, Z -5.5000, A 0.000, B 0.000, C 0.000 }
gfCNCPoint4[2846] = {X 358.3588, Y 69.5046, Z -5.5000, A 0.000, B 0.000, C 0.000 }
gfCNCPoint4[2847] = {X 357.3478, Y 68.1048, Z -5.5000, A 0.000, B 0.000, C 0.000 }
gfCNCPoint4[2848] = {X 356.4850, Y 66.6091, Z -5.5000, A 0.000, B 0.000, C 0.000 }
gfCNCPoint4[2849] = {X 355.7796, Y 65.0330, Z -5.5000, A 0.000, B 0.000, C 0.000 }
gfCNCPoint4[2850] = {X 355.2389, Y 63.3931, Z -5.5000, A 0.000, B 0.000, C 0.000 }
gfCNCPoint4[2851] = {X 354.8685, Y 61.7066, Z -5.5000, A 0.000, B 0.000, C 0.000 }
gfCNCPoint4[2852] = {X 352.1894, Y 62.2006, Z -5.5000, A 0.000, B 0.000, C 0.000 }
gfCNCPoint4[2853] = {X 349.4804, Y 62.4882, Z -5.5000, A 0.000, B 0.000, C 0.000 }
gfCNCPoint4[2854] = {X 349.3185, Y 60.0937, Z -5.5000, A 0.000, B 0.000, C 0.000 }
gfCNCPoint4[2855] = {X 348.2755, Y 60.1477, Z -5.5000, A 0.000, B 0.000, C 0.000 }
gfCNCPoint4[2856] = {X 347.2313, Y 60.1689, Z -5.5000, A 0.000, B 0.000, C 0.000 }
gfCNCPoint4[2857] = {X 344.3951, Y 60.1148, Z -5.5000, A 0.000, B 0.000, C 0.000 }
gfCNCPoint4[2858] = {X 341.5733, Y 59.8242, Z -5.5000, A 0.000, B 0.000, C 0.000 }
gfCNCPoint4[2859] = {X 338.7856, Y 59.2991, Z -5.5000, A 0.000, B 0.000, C 0.000 }
gfCNCPoint4[2860] = {X 338.6400, Y 60.9984, Z -5.5000, A 0.000, B 0.000, C 0.000 }
gfCNCPoint4[2861] = {X 338.2961, Y 62.6689, Z -5.5000, A 0.000, B 0.000, C 0.000 }
gfCNCPoint4[2862] = {X 337.7587, Y 64.2875, Z -5.5000, A 0.000, B 0.000, C 0.000 }
gfCNCPoint4[2863] = {X 337.0352, Y 65.8319, Z -5.5000, A 0.000, B 0.000, C 0.000 }
gfCNCPoint4[2864] = {X 336.1356, Y 67.2809, Z -5.5000, A 0.000, B 0.000, C 0.000 }
gfCNCPoint4[2865] = {X 335.0723, Y 68.6143, Z -5.5000, A 0.000, B 0.000, C 0.000 }
gfCNCPoint4[2866] = {X 335.0733, Y 79.5899, Z -5.5000, A 0.000, B 0.000, C 0.000 }
gfCNCPoint4[2867] = {X 335.9714, Y 79.6973, Z -5.5000, A 0.000, B 0.000, C 0.000 }
gfCNCPoint4[2868] = {X 336.8719, Y 79.7828, Z -5.5000, A 0.000, B 0.000, C 0.000 }
gfCNCPoint4[2869] = {X 340.9430, Y 80.0568, Z -5.5000, A 0.000, B 0.000, C 0.000 }
gfCNCPoint4[2870] = {X 345.0208, Y 80.1991, Z -5.5000, A 0.000, B 0.000, C 0.000 }
gfCNCPoint4[2871] = {X 349.1011, Y 80.2096, Z -5.5000, A 0.000, B 0.000, C 0.000 }
gfCNCPoint4[2872] = {X 352.9063, Y 80.1494, Z -5.5000, A 0.000, B 0.000, C 0.000 }
gfCNCPoint4[2873] = {X 356.7068, Y 79.9504, Z -5.5000, A 0.000, B 0.000, C 0.000 }
gfCNCPoint4[2874] = {X 360.4975, Y 79.6126, Z -5.5000, A 0.000, B 0.000, C 0.000 }
gfCNCPoint4[2875] = {X 360.7595, Y 79.5825, Z -5.5000, A 0.000, B 0.000, C 0.000 }
gfCNCPoint4[2876] = {X 360.7587, Y 68.6233, Z -5.5000, A 0.000, B 0.000, C 0.000 }
gfCNCPoint4[2877] = {X 359.7297, Y 67.3409, Z -5.5000, A 0.000, B 0.000, C 0.000 }
gfCNCPoint4[2878] = {X 358.8526, Y 65.9502, Z -5.5000, A 0.000, B 0.000, C 0.000 }
gfCNCPoint4[2879] = {X 358.1389, Y 64.4689, Z -5.5000, A 0.000, B 0.000, C 0.000 }
gfCNCPoint4[2880] = {X 357.5976, Y 62.9163, Z -5.5000, A 0.000, B 0.000, C 0.000 }
gfCNCPoint4[2881] = {X 357.2359, Y 61.3124, Z -5.5000, A 0.000, B 0.000, C 0.000 }
gfCNCPoint4[2882] = {X 357.0916, Y 60.1638, Z -5.5000, A 0.000, B 0.000, C 0.000 }
gfCNCPoint4[2883] = {X 357.0395, Y 59.0073, Z -5.5000, A 0.000, B 0.000, C 0.000 }
gfCNCPoint4[2884] = {X 357.0394, Y 58.6397, Z -5.5000, A 0.000, B 0.000, C 0.000 }
gfCNCPoint4[2885] = {X 355.6990, Y 59.0306, Z -5.5000, A 0.000, B 0.000, C 0.000 }
gfCNCPoint4[2886] = {X 354.3433, Y 59.3648, Z -5.5000, A 0.000, B 0.000, C 0.000 }
gfCNCPoint4[2887] = {X 351.8449, Y 59.8255, Z -5.5000, A 0.000, B 0.000, C 0.000 }
gfCNCPoint4[2888] = {X 349.3185, Y 60.0937, Z -5.5000, A 0.000, B 0.000, C 0.000 }
gfCNCPoint4[2889] = {X 349.1567, Y 57.6992, Z -5.5000, A 0.000, B 0.000, C 0.000 }
gfCNCPoint4[2890] = {X 348.1782, Y 57.7497, Z -5.5000, A 0.000, B 0.000, C 0.000 }
gfCNCPoint4[2891] = {X 347.1987, Y 57.7690, Z -5.5000, A 0.000, B 0.000, C 0.000 }
gfCNCPoint4[2892] = {X 344.5556, Y 57.7201, Z -5.5000, A 0.000, B 0.000, C 0.000 }
gfCNCPoint4[2893] = {X 341.9258, Y 57.4502, Z -5.5000, A 0.000, B 0.000, C 0.000 }
gfCNCPoint4[2894] = {X 339.3279, Y 56.9612, Z -5.5000, A 0.000, B 0.000, C 0.000 }
gfCNCPoint4[2895] = {X 337.7709, Y 56.5580, Z -5.5000, A 0.000, B 0.000, C 0.000 }
gfCNCPoint4[2896] = {X 336.2365, Y 56.0760, Z -5.5000, A 0.000, B 0.000, C 0.000 }
gfCNCPoint4[2897] = {X 336.3521, Y 57.0349, Z -5.5000, A 0.000, B 0.000, C 0.000 }
gfCNCPoint4[2898] = {X 336.3907, Y 58.0000, Z -5.5000, A 0.000, B 0.000, C 0.000 }
gfCNCPoint4[2899] = {X 336.3907, Y 58.9522, Z -5.5000, A 0.000, B 0.000, C 0.000 }
gfCNCPoint4[2900] = {X 336.3894, Y 59.0936, Z -5.5000, A 0.000, B 0.000, C 0.000 }
gfCNCPoint4[2901] = {X 336.3864, Y 59.2351, Z -5.5000, A 0.000, B 0.000, C 0.000 }
gfCNCPoint4[2902] = {X 336.2428, Y 60.7992, Z -5.5000, A 0.000, B 0.000, C 0.000 }
gfCNCPoint4[2903] = {X 335.8981, Y 62.3317, Z -5.5000, A 0.000, B 0.000, C 0.000 }
gfCNCPoint4[2904] = {X 335.3581, Y 63.8067, Z -5.5000, A 0.000, B 0.000, C 0.000 }
gfCNCPoint4[2905] = {X 334.6318, Y 65.1994, Z -5.5000, A 0.000, B 0.000, C 0.000 }
gfCNCPoint4[2906] = {X 333.7315, Y 66.4865, Z -5.5000, A 0.000, B 0.000, C 0.000 }
gfCNCPoint4[2907] = {X 332.6722, Y 67.6463, Z -5.5000, A 0.000, B 0.000, C 0.000 }
gfCNCPoint4[2908] = {X 332.6734, Y 81.6371, Z -5.5000, A 0.000, B 0.000, C 0.000 }
gfCNCPoint4[2909] = {X 334.6670, Y 81.9570, Z -5.5000, A 0.000, B 0.000, C 0.000 }
gfCNCPoint4[2910] = {X 336.6742, Y 82.1746, Z -5.5000, A 0.000, B 0.000, C 0.000 }
gfCNCPoint4[2911] = {X 340.8156, Y 82.4534, Z -5.5000, A 0.000, B 0.000, C 0.000 }
gfCNCPoint4[2912] = {X 344.9638, Y 82.5984, Z -5.5000, A 0.000, B 0.000, C 0.000 }
gfCNCPoint4[2913] = {X 349.1145, Y 82.6096, Z -5.5000, A 0.000, B 0.000, C 0.000 }
gfCNCPoint4[2914] = {X 353.0020, Y 82.5476, Z -5.5000, A 0.000, B 0.000, C 0.000 }
gfCNCPoint4[2915] = {X 356.8846, Y 82.3438, Z -5.5000, A 0.000, B 0.000, C 0.000 }
gfCNCPoint4[2916] = {X 360.7571, Y 81.9985, Z -5.5000, A 0.000, B 0.000, C 0.000 }
gfCNCPoint4[2917] = {X 361.9620, Y 81.8413, Z -5.5000, A 0.000, B 0.000, C 0.000 }
gfCNCPoint4[2918] = {X 363.1596, Y 81.6356, Z -5.5000, A 0.000, B 0.000, C 0.000 }
gfCNCPoint4[2919] = {X 363.1587, Y 67.6534, Z -5.5000, A 0.000, B 0.000, C 0.000 }
gfCNCPoint4[2920] = {X 362.0726, Y 66.4631, Z -5.5000, A 0.000, B 0.000, C 0.000 }
gfCNCPoint4[2921] = {X 361.1546, Y 65.1389, Z -5.5000, A 0.000, B 0.000, C 0.000 }
gfCNCPoint4[2922] = {X 360.4210, Y 63.7043, Z -5.5000, A 0.000, B 0.000, C 0.000 }
gfCNCPoint4[2923] = {X 359.8849, Y 62.1849, Z -5.5000, A 0.000, B 0.000, C 0.000 }
gfCNCPoint4[2924] = {X 359.5558, Y 60.6076, Z -5.5000, A 0.000, B 0.000, C 0.000 }
gfCNCPoint4[2925] = {X 359.4395, Y 59.0005, Z -5.5000, A 0.000, B 0.000, C 0.000 }
gfCNCPoint4[2926] = {X 359.4393, Y 58.0000, Z -5.5000, A 0.000, B 0.000, C 0.000 }
gfCNCPoint4[2927] = {X 359.5340, Y 56.4899, Z -5.5000, A 0.000, B 0.000, C 0.000 }
gfCNCPoint4[2928] = {X 359.8168, Y 55.0036, Z -5.5000, A 0.000, B 0.000, C 0.000 }
gfCNCPoint4[2929] = {X 359.6071, Y 55.1017, Z -5.5000, A 0.000, B 0.000, C 0.000 }
gfCNCPoint4[2930] = {X 359.3967, Y 55.1983, Z -5.5000, A 0.000, B 0.000, C 0.000 }
gfCNCPoint4[2931] = {X 357.8733, Y 55.8154, Z -5.5000, A 0.000, B 0.000, C 0.000 }
gfCNCPoint4[2932] = {X 356.3192, Y 56.3503, Z -5.5000, A 0.000, B 0.000, C 0.000 }
gfCNCPoint4[2933] = {X 353.9698, Y 56.9885, Z -5.5000, A 0.000, B 0.000, C 0.000 }
gfCNCPoint4[2934] = {X 351.5773, Y 57.4391, Z -5.5000, A 0.000, B 0.000, C 0.000 }
gfCNCPoint4[2935] = {X 349.1567, Y 57.6992, Z -5.5000, A 0.000, B 0.000, C 0.000 }
gfCNCPoint4[2936] = {X 348.9948, Y 55.3046, Z -5.5000, A 0.000, B 0.000, C 0.000 }
gfCNCPoint4[2937] = {X 348.0809, Y 55.3516, Z -5.5000, A 0.000, B 0.000, C 0.000 }
gfCNCPoint4[2938] = {X 347.1660, Y 55.3691, Z -5.5000, A 0.000, B 0.000, C 0.000 }
gfCNCPoint4[2939] = {X 344.5859, Y 55.3173, Z -5.5000, A 0.000, B 0.000, C 0.000 }
gfCNCPoint4[2940] = {X 342.0205, Y 55.0377, Z -5.5000, A 0.000, B 0.000, C 0.000 }
gfCNCPoint4[2941] = {X 339.4899, Y 54.5324, Z -5.5000, A 0.000, B 0.000, C 0.000 }
gfCNCPoint4[2942] = {X 337.0138, Y 53.8054, Z -5.5000, A 0.000, B 0.000, C 0.000 }
gfCNCPoint4[2943] = {X 334.7577, Y 52.9268, Z -5.5000, A 0.000, B 0.000, C 0.000 }
gfCNCPoint4[2944] = {X 332.5823, Y 51.8642, Z -5.5000, A 0.000, B 0.000, C 0.000 }
gfCNCPoint4[2945] = {X 331.5881, Y 51.2800, Z -5.5000, A 0.000, B 0.000, C 0.000 }
gfCNCPoint4[2946] = {X 330.6179, Y 50.6568, Z -5.5000, A 0.000, B 0.000, C 0.000 }
gfCNCPoint4[2947] = {X 331.5824, Y 51.6106, Z -5.5000, A 0.000, B 0.000, C 0.000 }
gfCNCPoint4[2948] = {X 332.4041, Y 52.6897, Z -5.5000, A 0.000, B 0.000, C 0.000 }
gfCNCPoint4[2949] = {X 333.0669, Y 53.8731, Z -5.5000, A 0.000, B 0.000, C 0.000 }
gfCNCPoint4[2950] = {X 333.5578, Y 55.1376, Z -5.5000, A 0.000, B 0.000, C 0.000 }
gfCNCPoint4[2951] = {X 333.8671, Y 56.4582, Z -5.5000, A 0.000, B 0.000, C 0.000 }
gfCNCPoint4[2952] = {X 333.9597, Y 57.2267, Z -5.5000, A 0.000, B 0.000, C 0.000 }
gfCNCPoint4[2953] = {X 333.9907, Y 58.0000, Z -5.5000, A 0.000, B 0.000, C 0.000 }
gfCNCPoint4[2954] = {X 333.9907, Y 58.9442, Z -5.5000, A 0.000, B 0.000, C 0.000 }
gfCNCPoint4[2955] = {X 333.8762, Y 60.3994, Z -5.5000, A 0.000, B 0.000, C 0.000 }
gfCNCPoint4[2956] = {X 333.5450, Y 61.8210, Z -5.5000, A 0.000, B 0.000, C 0.000 }
gfCNCPoint4[2957] = {X 333.0046, Y 63.1770, Z -5.5000, A 0.000, B 0.000, C 0.000 }
gfCNCPoint4[2958] = {X 332.2673, Y 64.4368, Z -5.5000, A 0.000, B 0.000, C 0.000 }
gfCNCPoint4[2959] = {X 331.3495, Y 65.5719, Z -5.5000, A 0.000, B 0.000, C 0.000 }
gfCNCPoint4[2960] = {X 330.2721, Y 66.5567, Z -5.5000, A 0.000, B 0.000, C 0.000 }
gfCNCPoint4[2961] = {X 330.2736, Y 83.2032, Z -5.5000, A 0.000, B 0.000, C 0.000 }
gfCNCPoint4[2962] = {X 330.2773, Y 83.5826, Z -5.5000, A 0.000, B 0.000, C 0.000 }
gfCNCPoint4[2963] = {X 333.3585, Y 84.1908, Z -5.5000, A 0.000, B 0.000, C 0.000 }
gfCNCPoint4[2964] = {X 336.4766, Y 84.5665, Z -5.5000, A 0.000, B 0.000, C 0.000 }
gfCNCPoint4[2965] = {X 340.6882, Y 84.8500, Z -5.5000, A 0.000, B 0.000, C 0.000 }
gfCNCPoint4[2966] = {X 344.9068, Y 84.9978, Z -5.5000, A 0.000, B 0.000, C 0.000 }
gfCNCPoint4[2967] = {X 349.1279, Y 85.0097, Z -5.5000, A 0.000, B 0.000, C 0.000 }
gfCNCPoint4[2968] = {X 353.0976, Y 84.9457, Z -5.5000, A 0.000, B 0.000, C 0.000 }
gfCNCPoint4[2969] = {X 357.0623, Y 84.7372, Z -5.5000, A 0.000, B 0.000, C 0.000 }
gfCNCPoint4[2970] = {X 361.0167, Y 84.3845, Z -5.5000, A 0.000, B 0.000, C 0.000 }
gfCNCPoint4[2971] = {X 363.3030, Y 84.0505, Z -5.5000, A 0.000, B 0.000, C 0.000 }
gfCNCPoint4[2972] = {X 365.5597, Y 83.5552, Z -5.5000, A 0.000, B 0.000, C 0.000 }
gfCNCPoint4[2973] = {X 365.5586, Y 66.5612, Z -5.5000, A 0.000, B 0.000, C 0.000 }
gfCNCPoint4[2974] = {X 364.4843, Y 65.5832, Z -5.5000, A 0.000, B 0.000, C 0.000 }
gfCNCPoint4[2975] = {X 363.5684, Y 64.4555, Z -5.5000, A 0.000, B 0.000, C 0.000 }
gfCNCPoint4[2976] = {X 362.8316, Y 63.2034, Z -5.5000, A 0.000, B 0.000, C 0.000 }
gfCNCPoint4[2977] = {X 362.2905, Y 61.8551, Z -5.5000, A 0.000, B 0.000, C 0.000 }
gfCNCPoint4[2978] = {X 361.9573, Y 60.4410, Z -5.5000, A 0.000, B 0.000, C 0.000 }
gfCNCPoint4[2979] = {X 361.8395, Y 58.9930, Z -5.5000, A 0.000, B 0.000, C 0.000 }
gfCNCPoint4[2980] = {X 361.8393, Y 58.0000, Z -5.5000, A 0.000, B 0.000, C 0.000 }
gfCNCPoint4[2981] = {X 361.9152, Y 56.7899, Z -5.5000, A 0.000, B 0.000, C 0.000 }
gfCNCPoint4[2982] = {X 362.1418, Y 55.5989, Z -5.5000, A 0.000, B 0.000, C 0.000 }
gfCNCPoint4[2983] = {X 362.5728, Y 54.3038, Z -5.5000, A 0.000, B 0.000, C 0.000 }
gfCNCPoint4[2984] = {X 363.1816, Y 53.0821, Z -5.5000, A 0.000, B 0.000, C 0.000 }
gfCNCPoint4[2985] = {X 363.9562, Y 51.9583, Z -5.5000, A 0.000, B 0.000, C 0.000 }
gfCNCPoint4[2986] = {X 364.8812, Y 50.9545, Z -5.5000, A 0.000, B 0.000, C 0.000 }
gfCNCPoint4[2987] = {X 365.9382, Y 50.0909, Z -5.5000, A 0.000, B 0.000, C 0.000 }
gfCNCPoint4[2988] = {X 367.1061, Y 49.3845, Z -5.5000, A 0.000, B 0.000, C 0.000 }
gfCNCPoint4[2989] = {X 368.3618, Y 48.8494, Z -5.5000, A 0.000, B 0.000, C 0.000 }
gfCNCPoint4[2990] = {X 369.6803, Y 48.4963, Z -5.5000, A 0.000, B 0.000, C 0.000 }
gfCNCPoint4[2991] = {X 371.0354, Y 48.3321, Z -5.5000, A 0.000, B 0.000, C 0.000 }
gfCNCPoint4[2992] = {X 371.2772, Y 48.3230, Z -5.5000, A 0.000, B 0.000, C 0.000 }
gfCNCPoint4[2993] = {X 371.5193, Y 48.3200, Z -5.5000, A 0.000, B 0.000, C 0.000 }
gfCNCPoint4[2994] = {X 388.0597, Y 48.3200, Z -5.5000, A 0.000, B 0.000, C 0.000 }
gfCNCPoint4[2995] = {X 389.4419, Y 48.4192, Z -5.5000, A 0.000, B 0.000, C 0.000 }
gfCNCPoint4[2996] = {X 390.7958, Y 48.7147, Z -5.5000, A 0.000, B 0.000, C 0.000 }
gfCNCPoint4[2997] = {X 392.0936, Y 49.2006, Z -5.5000, A 0.000, B 0.000, C 0.000 }
gfCNCPoint4[2998] = {X 393.3087, Y 49.8667, Z -5.5000, A 0.000, B 0.000, C 0.000 }
gfCNCPoint4[2999] = {X 394.5333, Y 49.1962, Z -5.5000, A 0.000, B 0.000, C 0.000 }
gfCNCPoint4[3000] = {X 395.8416, Y 48.7089, Z -5.5000, A 0.000, B 0.000, C 0.000 }
gfCNCPoint4[3001] = {X 397.1858, Y 48.4177, Z -5.5000, A 0.000, B 0.000, C 0.000 }
gfCNCPoint4[3002] = {X 398.5577, Y 48.3200, Z -5.5000, A 0.000, B 0.000, C 0.000 }
gfCNCPoint4[3003] = {X 398.7346, Y 48.3200, Z -5.5000, A 0.000, B 0.000, C 0.000 }
gfCNCPoint4[3004] = {X 398.1859, Y 47.6069, Z -5.5000, A 0.000, B 0.000, C 0.000 }
gfCNCPoint4[3005] = {X 397.7774, Y 46.8051, Z -5.5000, A 0.000, B 0.000, C 0.000 }
gfCNCPoint4[3006] = {X 397.5230, Y 45.9420, Z -5.5000, A 0.000, B 0.000, C 0.000 }
gfCNCPoint4[3007] = {X 397.4561, Y 45.4921, Z -5.5000, A 0.000, B 0.000, C 0.000 }
gfCNCPoint4[3008] = {X 397.4314, Y 45.0378, Z -5.5000, A 0.000, B 0.000, C 0.000 }
gfCNCPoint4[3009] = {X 397.4316, Y 44.1456, Z -5.5000, A 0.000, B 0.000, C 0.000 }
gfCNCPoint4[3010] = {X 397.5413, Y 43.1780, Z -5.5000, A 0.000, B 0.000, C 0.000 }
gfCNCPoint4[3011] = {X 397.8410, Y 42.2514, Z -5.5000, A 0.000, B 0.000, C 0.000 }
gfCNCPoint4[3012] = {X 398.3186, Y 41.4029, Z -5.5000, A 0.000, B 0.000, C 0.000 }
gfCNCPoint4[3013] = {X 398.9552, Y 40.6660, Z -5.5000, A 0.000, B 0.000, C 0.000 }
gfCNCPoint4[3014] = {X 398.9552, Y 31.8241, Z -5.5000, A 0.000, B 0.000, C 0.000 }
gfCNCPoint4[3015] = {X 393.0323, Y 21.5245, Z -5.5000, A 0.000, B 0.000, C 0.000 }
gfCNCPoint4[3016] = {X 392.1497, Y 20.0229, Z -5.5000, A 0.000, B 0.000, C 0.000 }
gfCNCPoint4[3017] = {X 391.2386, Y 18.5383, Z -5.5000, A 0.000, B 0.000, C 0.000 }
gfCNCPoint4[3018] = {X 390.8281, Y 17.9625, Z -5.5000, A 0.000, B 0.000, C 0.000 }
gfCNCPoint4[3019] = {X 390.3523, Y 17.4395, Z -5.5000, A 0.000, B 0.000, C 0.000 }
gfCNCPoint4[3020] = {X 389.5424, Y 16.9837, Z -5.5000, A 0.000, B 0.000, C 0.000 }
gfCNCPoint4[3021] = {X 388.8336, Y 16.3827, Z -5.5000, A 0.000, B 0.000, C 0.000 }
gfCNCPoint4[3022] = {X 388.2515, Y 15.6582, Z -5.5000, A 0.000, B 0.000, C 0.000 }
gfCNCPoint4[3023] = {X 387.8174, Y 14.8365, Z -5.5000, A 0.000, B 0.000, C 0.000 }
gfCNCPoint4[3024] = {X 387.5469, Y 13.9475, Z -5.5000, A 0.000, B 0.000, C 0.000 }
gfCNCPoint4[3025] = {X 387.4498, Y 13.0232, Z -5.5000, A 0.000, B 0.000, C 0.000 }
gfCNCPoint4[3026] = {X 387.4496, Y 12.1868, Z -5.5000, A 0.000, B 0.000, C 0.000 }
gfCNCPoint4[3027] = {X 387.5362, Y 11.2717, Z -5.5000, A 0.000, B 0.000, C 0.000 }
gfCNCPoint4[3028] = {X 387.7928, Y 10.3891, Z -5.5000, A 0.000, B 0.000, C 0.000 }
gfCNCPoint4[3029] = {X 388.2376, Y 9.5280, Z -5.5000, A 0.000, B 0.000, C 0.000 }
gfCNCPoint4[3030] = {X 388.8437, Y 8.7718, Z -5.5000, A 0.000, B 0.000, C 0.000 }
gfCNCPoint4[3031] = {X 389.5872, Y 8.1503, Z -5.5000, A 0.000, B 0.000, C 0.000 }
gfCNCPoint4[3032] = {X 390.4390, Y 7.6879, Z -5.5000, A 0.000, B 0.000, C 0.000 }
gfCNCPoint4[3033] = {X 391.3653, Y 7.4030, Z -5.5000, A 0.000, B 0.000, C 0.000 }
gfCNCPoint4[3034] = {X 392.3296, Y 7.3068, Z -5.5000, A 0.000, B 0.000, C 0.000 }
gfCNCPoint4[3035] = {X 399.1118, Y 7.3068, Z -5.5000, A 0.000, B 0.000, C 0.000 }
gfCNCPoint4[3036] = {X 400.0638, Y 7.4006, Z -5.5000, A 0.000, B 0.000, C 0.000 }
gfCNCPoint4[3037] = {X 400.9793, Y 7.6783, Z -5.5000, A 0.000, B 0.000, C 0.000 }
gfCNCPoint4[3038] = {X 401.8229, Y 8.1292, Z -5.5000, A 0.000, B 0.000, C 0.000 }
gfCNCPoint4[3039] = {X 402.5624, Y 8.7361, Z -5.5000, A 0.000, B 0.000, C 0.000 }
gfCNCPoint4[3040] = {X 403.1693, Y 9.4756, Z -5.5000, A 0.000, B 0.000, C 0.000 }
gfCNCPoint4[3041] = {X 403.6203, Y 10.3193, Z -5.5000, A 0.000, B 0.000, C 0.000 }
gfCNCPoint4[3042] = {X 403.8980, Y 11.2348, Z -5.5000, A 0.000, B 0.000, C 0.000 }
gfCNCPoint4[3043] = {X 403.9918, Y 12.1868, Z -5.5000, A 0.000, B 0.000, C 0.000 }
gfCNCPoint4[3044] = {X 403.9915, Y 13.0237, Z -5.5000, A 0.000, B 0.000, C 0.000 }
gfCNCPoint4[3045] = {X 403.9016, Y 13.9115, Z -5.5000, A 0.000, B 0.000, C 0.000 }
gfCNCPoint4[3046] = {X 403.6516, Y 14.7680, Z -5.5000, A 0.000, B 0.000, C 0.000 }
gfCNCPoint4[3047] = {X 405.3646, Y 17.7424, Z -5.5000, A 0.000, B 0.000, C 0.000 }
gfCNCPoint4[3048] = {X 407.2445, Y 14.6975, Z -5.5000, A 0.000, B 0.000, C 0.000 }
gfCNCPoint4[3049] = {X 407.0142, Y 13.8725, Z -5.5000, A 0.000, B 0.000, C 0.000 }
gfCNCPoint4[3050] = {X 406.9317, Y 13.0199, Z -5.5000, A 0.000, B 0.000, C 0.000 }
gfCNCPoint4[3051] = {X 406.9315, Y 12.1868, Z -5.5000, A 0.000, B 0.000, C 0.000 }
gfCNCPoint4[3052] = {X 407.0253, Y 11.2348, Z -5.5000, A 0.000, B 0.000, C 0.000 }
gfCNCPoint4[3053] = {X 407.3030, Y 10.3193, Z -5.5000, A 0.000, B 0.000, C 0.000 }
gfCNCPoint4[3054] = {X 407.7540, Y 9.4756, Z -5.5000, A 0.000, B 0.000, C 0.000 }
gfCNCPoint4[3055] = {X 408.3609, Y 8.7361, Z -5.5000, A 0.000, B 0.000, C 0.000 }
gfCNCPoint4[3056] = {X 409.1004, Y 8.1292, Z -5.5000, A 0.000, B 0.000, C 0.000 }
gfCNCPoint4[3057] = {X 409.9440, Y 7.6783, Z -5.5000, A 0.000, B 0.000, C 0.000 }
gfCNCPoint4[3058] = {X 410.8595, Y 7.4006, Z -5.5000, A 0.000, B 0.000, C 0.000 }
gfCNCPoint4[3059] = {X 411.8115, Y 7.3068, Z -5.5000, A 0.000, B 0.000, C 0.000 }
gfCNCPoint4[3060] = {X 419.3245, Y 7.3068, Z -5.5000, A 0.000, B 0.000, C 0.000 }
gfCNCPoint4[3061] = {X 420.2888, Y 7.4030, Z -5.5000, A 0.000, B 0.000, C 0.000 }
gfCNCPoint4[3062] = {X 421.2151, Y 7.6879, Z -5.5000, A 0.000, B 0.000, C 0.000 }
gfCNCPoint4[3063] = {X 422.0669, Y 8.1503, Z -5.5000, A 0.000, B 0.000, C 0.000 }
gfCNCPoint4[3064] = {X 422.8104, Y 8.7718, Z -5.5000, A 0.000, B 0.000, C 0.000 }
gfCNCPoint4[3065] = {X 423.4165, Y 9.5280, Z -5.5000, A 0.000, B 0.000, C 0.000 }
gfCNCPoint4[3066] = {X 423.8613, Y 10.3891, Z -5.5000, A 0.000, B 0.000, C 0.000 }
gfCNCPoint4[3067] = {X 424.1179, Y 11.2717, Z -5.5000, A 0.000, B 0.000, C 0.000 }
gfCNCPoint4[3068] = {X 424.2045, Y 12.1868, Z -5.5000, A 0.000, B 0.000, C 0.000 }
gfCNCPoint4[3069] = {X 424.2045, Y 12.9780, Z -5.5000, A 0.000, B 0.000, C 0.000 }
gfCNCPoint4[3070] = {X 424.1061, Y 13.9308, Z -5.5000, A 0.000, B 0.000, C 0.000 }
gfCNCPoint4[3071] = {X 423.8258, Y 14.8467, Z -5.5000, A 0.000, B 0.000, C 0.000 }
gfCNCPoint4[3072] = {X 423.3742, Y 15.6914, Z -5.5000, A 0.000, B 0.000, C 0.000 }
gfCNCPoint4[3073] = {X 422.7680, Y 16.4331, Z -5.5000, A 0.000, B 0.000, C 0.000 }
gfCNCPoint4[3074] = {X 422.0303, Y 17.0440, Z -5.5000, A 0.000, B 0.000, C 0.000 }
gfCNCPoint4[3075] = {X 421.1885, Y 17.5011, Z -5.5000, A 0.000, B 0.000, C 0.000 }
gfCNCPoint4[3076] = {X 420.5406, Y 18.3845, Z -5.5000, A 0.000, B 0.000, C 0.000 }
gfCNCPoint4[3077] = {X 419.9515, Y 19.3081, Z -5.5000, A 0.000, B 0.000, C 0.000 }
gfCNCPoint4[3078] = {X 414.1632, Y 28.6184, Z -5.5000, A 0.000, B 0.000, C 0.000 }
gfCNCPoint4[3079] = {X 422.3160, Y 33.6871, Z -5.5000, A 0.000, B 0.000, C 0.000 }
gfCNCPoint4[3080] = {X 421.8935, Y 34.3667, Z -5.5000, A 0.000, B 0.000, C 0.000 }
gfCNCPoint4[3081] = {X 422.1476, Y 34.0994, Z -5.5000, A 0.000, B 0.000, C 0.000 }
gfCNCPoint4[3082] = {X 422.4085, Y 33.8386, Z -5.5000, A 0.000, B 0.000, C 0.000 }
gfCNCPoint4[3083] = {X 422.3621, Y 33.7629, Z -5.5000, A 0.000, B 0.000, C 0.000 }
gfCNCPoint4[3084] = {X 422.3160, Y 33.6871, Z -5.5000, A 0.000, B 0.000, C 0.000 }
gfCNCPoint4[3085] = {X 420.2778, Y 32.4199, Z -5.5000, A 0.000, B 0.000, C 0.000 }
gfCNCPoint4[3086] = {X 419.3074, Y 33.9808, Z -5.5000, A 0.000, B 0.000, C 0.000 }
gfCNCPoint4[3087] = {X 419.3077, Y 38.3387, Z -5.5000, A 0.000, B 0.000, C 0.000 }
gfCNCPoint4[3088] = {X 419.9581, Y 39.7075, Z -5.5000, A 0.000, B 0.000, C 0.000 }
gfCNCPoint4[3089] = {X 420.4338, Y 41.1465, Z -5.5000, A 0.000, B 0.000, C 0.000 }
gfCNCPoint4[3090] = {X 420.6280, Y 41.1585, Z -5.5000, A 0.000, B 0.000, C 0.000 }
gfCNCPoint4[3091] = {X 420.8222, Y 41.1728, Z -5.5000, A 0.000, B 0.000, C 0.000 }
gfCNCPoint4[3092] = {X 421.2844, Y 39.7575, Z -5.5000, A 0.000, B 0.000, C 0.000 }
gfCNCPoint4[3093] = {X 421.9173, Y 38.4099, Z -5.5000, A 0.000, B 0.000, C 0.000 }
gfCNCPoint4[3094] = {X 422.7111, Y 37.1503, Z -5.5000, A 0.000, B 0.000, C 0.000 }
gfCNCPoint4[3095] = {X 423.6539, Y 35.9980, Z -5.5000, A 0.000, B 0.000, C 0.000 }
gfCNCPoint4[3096] = {X 424.3420, Y 35.3129, Z -5.5000, A 0.000, B 0.000, C 0.000 }
gfCNCPoint4[3097] = {X 425.0829, Y 34.6852, Z -5.5000, A 0.000, B 0.000, C 0.000 }
gfCNCPoint4[3098] = {X 425.4266, Y 34.0124, Z -5.5000, A 0.000, B 0.000, C 0.000 }
gfCNCPoint4[3099] = {X 424.8788, Y 33.2418, Z -5.5000, A 0.000, B 0.000, C 0.000 }
gfCNCPoint4[3100] = {X 424.3697, Y 32.4451, Z -5.5000, A 0.000, B 0.000, C 0.000 }
gfCNCPoint4[3101] = {X 423.3882, Y 30.6023, Z -5.5000, A 0.000, B 0.000, C 0.000 }
gfCNCPoint4[3102] = {X 422.6132, Y 28.6636, Z -5.5000, A 0.000, B 0.000, C 0.000 }
gfCNCPoint4[3103] = {X 420.2778, Y 32.4199, Z -5.5000, A 0.000, B 0.000, C 0.000 }
gfCNCPoint4[3104] = {X 418.2396, Y 31.1527, Z -5.5000, A 0.000, B 0.000, C 0.000 }
gfCNCPoint4[3105] = {X 416.9074, Y 33.2956, Z -5.5000, A 0.000, B 0.000, C 0.000 }
gfCNCPoint4[3106] = {X 416.9078, Y 38.9953, Z -5.5000, A 0.000, B 0.000, C 0.000 }
gfCNCPoint4[3107] = {X 417.4891, Y 40.0485, Z -5.5000, A 0.000, B 0.000, C 0.000 }
gfCNCPoint4[3108] = {X 417.9370, Y 41.1651, Z -5.5000, A 0.000, B 0.000, C 0.000 }
gfCNCPoint4[3109] = {X 418.2447, Y 42.3281, Z -5.5000, A 0.000, B 0.000, C 0.000 }
gfCNCPoint4[3110] = {X 418.4077, Y 43.5200, Z -5.5000, A 0.000, B 0.000, C 0.000 }
gfCNCPoint4[3111] = {X 419.4886, Y 43.5200, Z -5.5000, A 0.000, B 0.000, C 0.000 }
gfCNCPoint4[3112] = {X 421.1752, Y 43.6186, Z -5.5000, A 0.000, B 0.000, C 0.000 }
gfCNCPoint4[3113] = {X 422.8389, Y 43.9129, Z -5.5000, A 0.000, B 0.000, C 0.000 }
gfCNCPoint4[3114] = {X 423.0005, Y 42.4234, Z -5.5000, A 0.000, B 0.000, C 0.000 }
gfCNCPoint4[3115] = {X 423.3900, Y 40.9766, Z -5.5000, A 0.000, B 0.000, C 0.000 }
gfCNCPoint4[3116] = {X 423.9980, Y 39.6073, Z -5.5000, A 0.000, B 0.000, C 0.000 }
gfCNCPoint4[3117] = {X 424.8102, Y 38.3482, Z -5.5000, A 0.000, B 0.000, C 0.000 }
gfCNCPoint4[3118] = {X 425.8068, Y 37.2295, Z -5.5000, A 0.000, B 0.000, C 0.000 }
gfCNCPoint4[3119] = {X 426.9642, Y 36.2780, Z -5.5000, A 0.000, B 0.000, C 0.000 }
gfCNCPoint4[3120] = {X 428.2772, Y 33.7080, Z -5.5000, A 0.000, B 0.000, C 0.000 }
gfCNCPoint4[3121] = {X 427.2129, Y 32.3913, Z -5.5000, A 0.000, B 0.000, C 0.000 }
gfCNCPoint4[3122] = {X 426.2871, Y 30.9738, Z -5.5000, A 0.000, B 0.000, C 0.000 }
gfCNCPoint4[3123] = {X 425.5092, Y 29.4701, Z -5.5000, A 0.000, B 0.000, C 0.000 }
gfCNCPoint4[3124] = {X 424.8870, Y 27.8956, Z -5.5000, A 0.000, B 0.000, C 0.000 }
gfCNCPoint4[3125] = {X 424.6540, Y 27.1487, Z -5.5000, A 0.000, B 0.000, C 0.000 }
gfCNCPoint4[3126] = {X 424.4562, Y 26.3919, Z -5.5000, A 0.000, B 0.000, C 0.000 }
gfCNCPoint4[3127] = {X 424.0553, Y 24.2628, Z -5.5000, A 0.000, B 0.000, C 0.000 }
gfCNCPoint4[3128] = {X 423.8649, Y 22.1047, Z -5.5000, A 0.000, B 0.000, C 0.000 }
gfCNCPoint4[3129] = {X 418.2396, Y 31.1527, Z -5.5000, A 0.000, B 0.000, C 0.000 }
gfCNCPoint4[3130] = {X 416.2014, Y 29.8856, Z -5.5000, A 0.000, B 0.000, C 0.000 }
gfCNCPoint4[3131] = {X 414.5073, Y 32.6104, Z -5.5000, A 0.000, B 0.000, C 0.000 }
gfCNCPoint4[3132] = {X 414.5078, Y 39.7467, Z -5.5000, A 0.000, B 0.000, C 0.000 }
gfCNCPoint4[3133] = {X 415.1564, Y 40.7518, Z -5.5000, A 0.000, B 0.000, C 0.000 }
gfCNCPoint4[3134] = {X 415.6347, Y 41.8484, Z -5.5000, A 0.000, B 0.000, C 0.000 }
gfCNCPoint4[3135] = {X 415.9300, Y 43.0076, Z -5.5000, A 0.000, B 0.000, C 0.000 }
gfCNCPoint4[3136] = {X 416.0347, Y 44.1992, Z -5.5000, A 0.000, B 0.000, C 0.000 }
gfCNCPoint4[3137] = {X 416.0347, Y 45.0000, Z -5.5000, A 0.000, B 0.000, C 0.000 }
gfCNCPoint4[3138] = {X 416.0201, Y 45.4609, Z -5.5000, A 0.000, B 0.000, C 0.000 }
gfCNCPoint4[3139] = {X 415.9763, Y 45.9200, Z -5.5000, A 0.000, B 0.000, C 0.000 }
gfCNCPoint4[3140] = {X 419.4886, Y 45.9200, Z -5.5000, A 0.000, B 0.000, C 0.000 }
gfCNCPoint4[3141] = {X 420.8957, Y 46.0022, Z -5.5000, A 0.000, B 0.000, C 0.000 }
gfCNCPoint4[3142] = {X 422.2836, Y 46.2478, Z -5.5000, A 0.000, B 0.000, C 0.000 }
gfCNCPoint4[3143] = {X 423.4822, Y 46.5992, Z -5.5000, A 0.000, B 0.000, C 0.000 }
gfCNCPoint4[3144] = {X 424.6380, Y 47.0725, Z -5.5000, A 0.000, B 0.000, C 0.000 }
gfCNCPoint4[3145] = {X 425.7388, Y 47.6626, Z -5.5000, A 0.000, B 0.000, C 0.000 }
gfCNCPoint4[3146] = {X 425.4600, Y 46.7984, Z -5.5000, A 0.000, B 0.000, C 0.000 }
gfCNCPoint4[3147] = {X 425.2910, Y 45.9063, Z -5.5000, A 0.000, B 0.000, C 0.000 }
gfCNCPoint4[3148] = {X 425.2344, Y 45.0000, Z -5.5000, A 0.000, B 0.000, C 0.000 }
gfCNCPoint4[3149] = {X 425.2344, Y 44.2089, Z -5.5000, A 0.000, B 0.000, C 0.000 }
gfCNCPoint4[3150] = {X 425.2353, Y 44.0976, Z -5.5000, A 0.000, B 0.000, C 0.000 }
gfCNCPoint4[3151] = {X 425.2378, Y 43.9863, Z -5.5000, A 0.000, B 0.000, C 0.000 }
gfCNCPoint4[3152] = {X 425.3770, Y 42.7748, Z -5.5000, A 0.000, B 0.000, C 0.000 }
gfCNCPoint4[3153] = {X 425.7165, Y 41.6036, Z -5.5000, A 0.000, B 0.000, C 0.000 }
gfCNCPoint4[3154] = {X 426.2468, Y 40.5054, Z -5.5000, A 0.000, B 0.000, C 0.000 }
gfCNCPoint4[3155] = {X 426.9528, Y 39.5112, Z -5.5000, A 0.000, B 0.000, C 0.000 }
gfCNCPoint4[3156] = {X 427.8150, Y 38.6488, Z -5.5000, A 0.000, B 0.000, C 0.000 }
gfCNCPoint4[3157] = {X 428.8090, Y 37.9424, Z -5.5000, A 0.000, B 0.000, C 0.000 }
gfCNCPoint4[3158] = {X 431.2078, Y 33.2470, Z -5.5000, A 0.000, B 0.000, C 0.000 }
gfCNCPoint4[3159] = {X 429.9738, Y 32.0040, Z -5.5000, A 0.000, B 0.000, C 0.000 }
gfCNCPoint4[3160] = {X 428.9004, Y 30.6200, Z -5.5000, A 0.000, B 0.000, C 0.000 }
gfCNCPoint4[3161] = {X 428.0037, Y 29.1154, Z -5.5000, A 0.000, B 0.000, C 0.000 }
gfCNCPoint4[3162] = {X 427.2971, Y 27.5128, Z -5.5000, A 0.000, B 0.000, C 0.000 }
gfCNCPoint4[3163] = {X 426.7910, Y 25.8360, Z -5.5000, A 0.000, B 0.000, C 0.000 }
gfCNCPoint4[3164] = {X 426.4331, Y 23.9366, Z -5.5000, A 0.000, B 0.000, C 0.000 }
gfCNCPoint4[3165] = {X 426.2631, Y 22.0113, Z -5.5000, A 0.000, B 0.000, C 0.000 }
gfCNCPoint4[3166] = {X 426.2912, Y 19.9439, Z -5.5000, A 0.000, B 0.000, C 0.000 }
gfCNCPoint4[3167] = {X 426.5358, Y 17.8909, Z -5.5000, A 0.000, B 0.000, C 0.000 }
gfCNCPoint4[3168] = {X 426.9943, Y 15.8749, Z -5.5000, A 0.000, B 0.000, C 0.000 }
gfCNCPoint4[3169] = {X 427.6129, Y 14.1191, Z -5.5000, A 0.000, B 0.000, C 0.000 }
gfCNCPoint4[3170] = {X 428.4472, Y 12.4549, Z -5.5000, A 0.000, B 0.000, C 0.000 }
gfCNCPoint4[3171] = {X 429.4839, Y 10.9087, Z -5.5000, A 0.000, B 0.000, C 0.000 }
gfCNCPoint4[3172] = {X 430.7066, Y 9.5049, Z -5.5000, A 0.000, B 0.000, C 0.000 }
gfCNCPoint4[3173] = {X 426.0925, Y 9.5049, Z -5.5000, A 0.000, B 0.000, C 0.000 }
gfCNCPoint4[3174] = {X 426.3754, Y 10.3750, Z -5.5000, A 0.000, B 0.000, C 0.000 }
gfCNCPoint4[3175] = {X 426.5470, Y 11.2737, Z -5.5000, A 0.000, B 0.000, C 0.000 }
gfCNCPoint4[3176] = {X 426.6045, Y 12.1868, Z -5.5000, A 0.000, B 0.000, C 0.000 }
gfCNCPoint4[3177] = {X 426.6044, Y 12.9919, Z -5.5000, A 0.000, B 0.000, C 0.000 }
gfCNCPoint4[3178] = {X 426.4806, Y 14.2926, Z -5.5000, A 0.000, B 0.000, C 0.000 }
gfCNCPoint4[3179] = {X 426.1282, Y 15.5508, Z -5.5000, A 0.000, B 0.000, C 0.000 }
gfCNCPoint4[3180] = {X 425.5584, Y 16.7267, Z -5.5000, A 0.000, B 0.000, C 0.000 }
gfCNCPoint4[3181] = {X 424.7892, Y 17.7829, Z -5.5000, A 0.000, B 0.000, C 0.000 }
gfCNCPoint4[3182] = {X 423.8450, Y 18.6860, Z -5.5000, A 0.000, B 0.000, C 0.000 }
gfCNCPoint4[3183] = {X 422.7557, Y 19.4075, Z -5.5000, A 0.000, B 0.000, C 0.000 }
gfCNCPoint4[3184] = {X 422.3658, Y 19.9717, Z -5.5000, A 0.000, B 0.000, C 0.000 }
gfCNCPoint4[3185] = {X 422.0031, Y 20.5538, Z -5.5000, A 0.000, B 0.000, C 0.000 }
gfCNCPoint4[3186] = {X 416.2014, Y 29.8856, Z -5.5000, A 0.000, B 0.000, C 0.000 }
gfCNCPoint4[3187] = {X 414.1632, Y 28.6184, Z -5.5000, A 0.000, B 0.000, C 0.000 }
gfCNCPoint4[3188] = {X 412.1073, Y 31.9253, Z -5.5000, A 0.000, B 0.000, C 0.000 }
gfCNCPoint4[3189] = {X 412.1079, Y 40.6517, Z -5.5000, A 0.000, B 0.000, C 0.000 }
gfCNCPoint4[3190] = {X 412.7496, Y 41.4082, Z -5.5000, A 0.000, B 0.000, C 0.000 }
gfCNCPoint4[3191] = {X 413.2294, Y 42.2766, Z -5.5000, A 0.000, B 0.000, C 0.000 }
gfCNCPoint4[3192] = {X 413.5284, Y 43.2225, Z -5.5000, A 0.000, B 0.000, C 0.000 }
gfCNCPoint4[3193] = {X 413.6347, Y 44.2089, Z -5.5000, A 0.000, B 0.000, C 0.000 }
gfCNCPoint4[3194] = {X 413.6347, Y 45.0000, Z -5.5000, A 0.000, B 0.000, C 0.000 }
gfCNCPoint4[3195] = {X 413.6249, Y 45.3090, Z -5.5000, A 0.000, B 0.000, C 0.000 }
gfCNCPoint4[3196] = {X 413.5956, Y 45.6167, Z -5.5000, A 0.000, B 0.000, C 0.000 }
gfCNCPoint4[3197] = {X 413.3652, Y 46.5992, Z -5.5000, A 0.000, B 0.000, C 0.000 }
gfCNCPoint4[3198] = {X 412.9377, Y 47.5134, Z -5.5000, A 0.000, B 0.000, C 0.000 }
gfCNCPoint4[3199] = {X 412.3313, Y 48.3200, Z -5.5000, A 0.000, B 0.000, C 0.000 }
gfCNCPoint4[3200] = {X 411.9795, Y 47.9934, Z -5.5000, A 0.000, B 0.000, C 0.000 }
gfCNCPoint4[3201] = {X 411.3003, Y 48.5889, Z -5.5000, A 0.000, B 0.000, C 0.000 }
gfCNCPoint4[3202] = {X 410.5138, Y 49.0331, Z -5.5000, A 0.000, B 0.000, C 0.000 }
gfCNCPoint4[3203] = {X 409.6532, Y 49.3073, Z -5.5000, A 0.000, B 0.000, C 0.000 }
gfCNCPoint4[3204] = {X 408.7547, Y 49.4000, Z -5.5000, A 0.000, B 0.000, C 0.000 }
gfCNCPoint4[3205] = {X 402.3112, Y 49.4000, Z -5.5000, A 0.000, B 0.000, C 0.000 }
gfCNCPoint4[3206] = {X 401.3321, Y 49.2897, Z -5.5000, A 0.000, B 0.000, C 0.000 }
gfCNCPoint4[3207] = {X 400.4021, Y 48.9643, Z -5.5000, A 0.000, B 0.000, C 0.000 }
gfCNCPoint4[3208] = {X 399.5678, Y 48.4400, Z -5.5000, A 0.000, B 0.000, C 0.000 }
gfCNCPoint4[3209] = {X 398.8711, Y 47.7433, Z -5.5000, A 0.000, B 0.000, C 0.000 }
gfCNCPoint4[3210] = {X 398.3469, Y 46.9091, Z -5.5000, A 0.000, B 0.000, C 0.000 }
gfCNCPoint4[3211] = {X 398.0215, Y 45.9791, Z -5.5000, A 0.000, B 0.000, C 0.000 }
gfCNCPoint4[3212] = {X 397.9112, Y 45.0000, Z -5.5000, A 0.000, B 0.000, C 0.000 }
gfCNCPoint4[3213] = {X 397.9116, Y 44.1518, Z -5.5000, A 0.000, B 0.000, C 0.000 }
gfCNCPoint4[3214] = {X 398.0215, Y 43.2300, Z -5.5000, A 0.000, B 0.000, C 0.000 }
gfCNCPoint4[3215] = {X 398.3223, Y 42.3519, Z -5.5000, A 0.000, B 0.000, C 0.000 }
gfCNCPoint4[3216] = {X 398.8006, Y 41.5563, Z -5.5000, A 0.000, B 0.000, C 0.000 }
gfCNCPoint4[3217] = {X 399.4352, Y 40.8789, Z -5.5000, A 0.000, B 0.000, C 0.000 }
gfCNCPoint4[3218] = {X 399.4352, Y 31.6959, Z -5.5000, A 0.000, B 0.000, C 0.000 }
gfCNCPoint4[3219] = {X 393.4485, Y 21.2852, Z -5.5000, A 0.000, B 0.000, C 0.000 }
gfCNCPoint4[3220] = {X 392.5612, Y 19.7757, Z -5.5000, A 0.000, B 0.000, C 0.000 }
gfCNCPoint4[3221] = {X 391.6453, Y 18.2834, Z -5.5000, A 0.000, B 0.000, C 0.000 }
gfCNCPoint4[3222] = {X 391.1732, Y 17.6262, Z -5.5000, A 0.000, B 0.000, C 0.000 }
gfCNCPoint4[3223] = {X 390.6225, Y 17.0333, Z -5.5000, A 0.000, B 0.000, C 0.000 }
gfCNCPoint4[3224] = {X 389.8676, Y 16.6247, Z -5.5000, A 0.000, B 0.000, C 0.000 }
gfCNCPoint4[3225] = {X 389.2064, Y 16.0773, Z -5.5000, A 0.000, B 0.000, C 0.000 }
gfCNCPoint4[3226] = {X 388.6641, Y 15.4120, Z -5.5000, A 0.000, B 0.000, C 0.000 }
gfCNCPoint4[3227] = {X 388.2613, Y 14.6540, Z -5.5000, A 0.000, B 0.000, C 0.000 }
gfCNCPoint4[3228] = {X 388.0133, Y 13.8322, Z -5.5000, A 0.000, B 0.000, C 0.000 }
gfCNCPoint4[3229] = {X 387.9296, Y 12.9779, Z -5.5000, A 0.000, B 0.000, C 0.000 }
gfCNCPoint4[3230] = {X 387.9296, Y 12.1868, Z -5.5000, A 0.000, B 0.000, C 0.000 }
gfCNCPoint4[3231] = {X 388.0399, Y 11.2077, Z -5.5000, A 0.000, B 0.000, C 0.000 }
gfCNCPoint4[3232] = {X 388.3654, Y 10.2777, Z -5.5000, A 0.000, B 0.000, C 0.000 }
gfCNCPoint4[3233] = {X 388.8896, Y 9.4435, Z -5.5000, A 0.000, B 0.000, C 0.000 }
gfCNCPoint4[3234] = {X 389.5863, Y 8.7468, Z -5.5000, A 0.000, B 0.000, C 0.000 }
gfCNCPoint4[3235] = {X 390.4205, Y 8.2226, Z -5.5000, A 0.000, B 0.000, C 0.000 }
gfCNCPoint4[3236] = {X 391.3505, Y 7.8971, Z -5.5000, A 0.000, B 0.000, C 0.000 }
gfCNCPoint4[3237] = {X 392.3296, Y 7.7868, Z -5.5000, A 0.000, B 0.000, C 0.000 }
gfCNCPoint4[3238] = {X 399.1118, Y 7.7868, Z -5.5000, A 0.000, B 0.000, C 0.000 }
gfCNCPoint4[3239] = {X 400.0909, Y 7.8971, Z -5.5000, A 0.000, B 0.000, C 0.000 }
gfCNCPoint4[3240] = {X 401.0208, Y 8.2226, Z -5.5000, A 0.000, B 0.000, C 0.000 }
gfCNCPoint4[3241] = {X 401.8551, Y 8.7468, Z -5.5000, A 0.000, B 0.000, C 0.000 }
gfCNCPoint4[3242] = {X 402.5518, Y 9.4435, Z -5.5000, A 0.000, B 0.000, C 0.000 }
gfCNCPoint4[3243] = {X 403.0760, Y 10.2777, Z -5.5000, A 0.000, B 0.000, C 0.000 }
gfCNCPoint4[3244] = {X 403.4014, Y 11.2077, Z -5.5000, A 0.000, B 0.000, C 0.000 }
gfCNCPoint4[3245] = {X 403.5118, Y 12.1868, Z -5.5000, A 0.000, B 0.000, C 0.000 }
gfCNCPoint4[3246] = {X 403.5115, Y 13.0233, Z -5.5000, A 0.000, B 0.000, C 0.000 }
gfCNCPoint4[3247] = {X 403.4070, Y 13.9326, Z -5.5000, A 0.000, B 0.000, C 0.000 }
gfCNCPoint4[3248] = {X 403.1165, Y 14.8007, Z -5.5000, A 0.000, B 0.000, C 0.000 }
gfCNCPoint4[3249] = {X 405.3503, Y 18.6794, Z -5.5000, A 0.000, B 0.000, C 0.000 }
gfCNCPoint4[3250] = {X 407.7808, Y 14.7425, Z -5.5000, A 0.000, B 0.000, C 0.000 }
gfCNCPoint4[3251] = {X 407.5048, Y 13.8793, Z -5.5000, A 0.000, B 0.000, C 0.000 }
gfCNCPoint4[3252] = {X 407.4115, Y 12.9780, Z -5.5000, A 0.000, B 0.000, C 0.000 }
gfCNCPoint4[3253] = {X 407.4115, Y 12.1868, Z -5.5000, A 0.000, B 0.000, C 0.000 }
gfCNCPoint4[3254] = {X 407.5219, Y 11.2077, Z -5.5000, A 0.000, B 0.000, C 0.000 }
gfCNCPoint4[3255] = {X 407.8473, Y 10.2777, Z -5.5000, A 0.000, B 0.000, C 0.000 }
gfCNCPoint4[3256] = {X 408.3715, Y 9.4435, Z -5.5000, A 0.000, B 0.000, C 0.000 }
gfCNCPoint4[3257] = {X 409.0682, Y 8.7468, Z -5.5000, A 0.000, B 0.000, C 0.000 }
gfCNCPoint4[3258] = {X 409.9024, Y 8.2226, Z -5.5000, A 0.000, B 0.000, C 0.000 }
gfCNCPoint4[3259] = {X 410.8324, Y 7.8971, Z -5.5000, A 0.000, B 0.000, C 0.000 }
gfCNCPoint4[3260] = {X 411.8115, Y 7.7868, Z -5.5000, A 0.000, B 0.000, C 0.000 }
gfCNCPoint4[3261] = {X 419.3245, Y 7.7868, Z -5.5000, A 0.000, B 0.000, C 0.000 }
gfCNCPoint4[3262] = {X 420.3036, Y 7.8971, Z -5.5000, A 0.000, B 0.000, C 0.000 }
gfCNCPoint4[3263] = {X 421.2335, Y 8.2226, Z -5.5000, A 0.000, B 0.000, C 0.000 }
gfCNCPoint4[3264] = {X 422.0678, Y 8.7468, Z -5.5000, A 0.000, B 0.000, C 0.000 }
gfCNCPoint4[3265] = {X 422.7645, Y 9.4435, Z -5.5000, A 0.000, B 0.000, C 0.000 }
gfCNCPoint4[3266] = {X 423.2887, Y 10.2777, Z -5.5000, A 0.000, B 0.000, C 0.000 }
gfCNCPoint4[3267] = {X 423.6141, Y 11.2077, Z -5.5000, A 0.000, B 0.000, C 0.000 }
gfCNCPoint4[3268] = {X 423.7245, Y 12.1868, Z -5.5000, A 0.000, B 0.000, C 0.000 }
gfCNCPoint4[3269] = {X 423.7245, Y 12.9808, Z -5.5000, A 0.000, B 0.000, C 0.000 }
gfCNCPoint4[3270] = {X 423.6307, Y 13.8596, Z -5.5000, A 0.000, B 0.000, C 0.000 }
gfCNCPoint4[3271] = {X 423.3656, Y 14.7028, Z -5.5000, A 0.000, B 0.000, C 0.000 }
gfCNCPoint4[3272] = {X 422.9396, Y 15.4771, Z -5.5000, A 0.000, B 0.000, C 0.000 }
gfCNCPoint4[3273] = {X 422.3693, Y 16.1523, Z -5.5000, A 0.000, B 0.000, C 0.000 }
gfCNCPoint4[3274] = {X 421.6772, Y 16.7019, Z -5.5000, A 0.000, B 0.000, C 0.000 }
gfCNCPoint4[3275] = {X 420.8903, Y 17.1043, Z -5.5000, A 0.000, B 0.000, C 0.000 }
gfCNCPoint4[3276] = {X 420.1833, Y 18.0570, Z -5.5000, A 0.000, B 0.000, C 0.000 }
gfCNCPoint4[3277] = {X 419.5432, Y 19.0559, Z -5.5000, A 0.000, B 0.000, C 0.000 }
gfCNCPoint4[3278] = {X 418.0618, Y 21.4541, Z -5.5000, A 0.000, B 0.000, C 0.000 }
gfCNCPoint4[3279] = {X 411.6273, Y 31.7881, Z -5.5000, A 0.000, B 0.000, C 0.000 }
gfCNCPoint4[3280] = {X 411.6279, Y 40.8616, Z -5.5000, A 0.000, B 0.000, C 0.000 }
gfCNCPoint4[3281] = {X 412.2670, Y 41.5584, Z -5.5000, A 0.000, B 0.000, C 0.000 }
gfCNCPoint4[3282] = {X 412.7472, Y 42.3729, Z -5.5000, A 0.000, B 0.000, C 0.000 }
gfCNCPoint4[3283] = {X 413.0475, Y 43.2694, Z -5.5000, A 0.000, B 0.000, C 0.000 }
gfCNCPoint4[3284] = {X 413.1547, Y 44.2089, Z -5.5000, A 0.000, B 0.000, C 0.000 }
gfCNCPoint4[3285] = {X 413.1545, Y 45.0423, Z -5.5000, A 0.000, B 0.000, C 0.000 }
gfCNCPoint4[3286] = {X 413.0719, Y 45.8494, Z -5.5000, A 0.000, B 0.000, C 0.000 }
gfCNCPoint4[3287] = {X 412.8426, Y 46.6276, Z -5.5000, A 0.000, B 0.000, C 0.000 }
gfCNCPoint4[3288] = {X 412.4743, Y 47.3505, Z -5.5000, A 0.000, B 0.000, C 0.000 }
gfCNCPoint4[3289] = {X 411.9795, Y 47.9934, Z -5.5000, A 0.000, B 0.000, C 0.000 }
gfCNCPoint4[3290] = {X 412.3313, Y 48.3200, Z -5.5000, A 0.000, B 0.000, C 0.000 }
gfCNCPoint4[3291] = {X 419.4886, Y 48.3200, Z -5.5000, A 0.000, B 0.000, C 0.000 }
gfCNCPoint4[3292] = {X 420.8006, Y 48.4093, Z -5.5000, A 0.000, B 0.000, C 0.000 }
gfCNCPoint4[3293] = {X 422.0883, Y 48.6756, Z -5.5000, A 0.000, B 0.000, C 0.000 }
gfCNCPoint4[3294] = {X 423.3281, Y 49.1140, Z -5.5000, A 0.000, B 0.000, C 0.000 }
gfCNCPoint4[3295] = {X 424.4970, Y 49.7164, Z -5.5000, A 0.000, B 0.000, C 0.000 }
gfCNCPoint4[3296] = {X 425.4625, Y 50.3832, Z -5.5000, A 0.000, B 0.000, C 0.000 }
gfCNCPoint4[3297] = {X 426.3402, Y 51.1620, Z -5.5000, A 0.000, B 0.000, C 0.000 }
gfCNCPoint4[3298] = {X 427.1172, Y 52.0412, Z -5.5000, A 0.000, B 0.000, C 0.000 }
gfCNCPoint4[3299] = {X 427.7821, Y 53.0080, Z -5.5000, A 0.000, B 0.000, C 0.000 }
gfCNCPoint4[3300] = {X 428.1266, Y 53.6312, Z -5.5000, A 0.000, B 0.000, C 0.000 }
gfCNCPoint4[3301] = {X 428.4244, Y 54.2780, Z -5.5000, A 0.000, B 0.000, C 0.000 }
gfCNCPoint4[3302] = {X 431.5822, Y 55.5084, Z -5.5000, A 0.000, B 0.000, C 0.000 }
gfCNCPoint4[3303] = {X 439.8787, Y 58.8002, Z -5.5000, A 0.000, B 0.000, C 0.000 }
gfCNCPoint4[3304] = {X 441.6489, Y 54.3385, Z -5.5000, A 0.000, B 0.000, C 0.000 }
gfCNCPoint4[3305] = {X 444.2224, Y 55.3596, Z -5.5000, A 0.000, B 0.000, C 0.000 }
gfCNCPoint4[3306] = {X 444.5426, Y 54.0015, Z -5.5000, A 0.000, B 0.000, C 0.000 }
gfCNCPoint4[3307] = {X 444.9921, Y 52.6806, Z -5.5000, A 0.000, B 0.000, C 0.000 }
gfCNCPoint4[3308] = {X 443.9525, Y 53.3762, Z -5.5000, A 0.000, B 0.000, C 0.000 }
gfCNCPoint4[3309] = {X 442.8318, Y 53.9319, Z -5.5000, A 0.000, B 0.000, C 0.000 }
gfCNCPoint4[3310] = {X 441.6489, Y 54.3385, Z -5.5000, A 0.000, B 0.000, C 0.000 }
gfCNCPoint4[3311] = {X 440.7638, Y 56.5693, Z -5.5000, A 0.000, B 0.000, C 0.000 }
gfCNCPoint4[3312] = {X 446.3797, Y 58.7975, Z -5.5000, A 0.000, B 0.000, C 0.000 }
gfCNCPoint4[3313] = {X 446.3796, Y 58.0000, Z -5.5000, A 0.000, B 0.000, C 0.000 }
gfCNCPoint4[3314] = {X 446.4303, Y 56.8940, Z -5.5000, A 0.000, B 0.000, C 0.000 }
gfCNCPoint4[3315] = {X 446.5821, Y 55.7972, Z -5.5000, A 0.000, B 0.000, C 0.000 }
gfCNCPoint4[3316] = {X 446.8493, Y 54.6642, Z -5.5000, A 0.000, B 0.000, C 0.000 }
gfCNCPoint4[3317] = {X 447.2243, Y 53.5622, Z -5.5000, A 0.000, B 0.000, C 0.000 }
gfCNCPoint4[3318] = {X 447.8767, Y 52.1752, Z -5.5000, A 0.000, B 0.000, C 0.000 }
gfCNCPoint4[3319] = {X 448.6995, Y 50.8820, Z -5.5000, A 0.000, B 0.000, C 0.000 }
gfCNCPoint4[3320] = {X 447.8224, Y 50.1272, Z -5.5000, A 0.000, B 0.000, C 0.000 }
gfCNCPoint4[3321] = {X 447.0760, Y 49.2431, Z -5.5000, A 0.000, B 0.000, C 0.000 }
gfCNCPoint4[3322] = {X 446.4792, Y 48.2518, Z -5.5000, A 0.000, B 0.000, C 0.000 }
gfCNCPoint4[3323] = {X 446.0469, Y 47.1785, Z -5.5000, A 0.000, B 0.000, C 0.000 }
gfCNCPoint4[3324] = {X 445.6333, Y 48.2126, Z -5.5000, A 0.000, B 0.000, C 0.000 }
gfCNCPoint4[3325] = {X 445.0668, Y 49.1715, Z -5.5000, A 0.000, B 0.000, C 0.000 }
gfCNCPoint4[3326] = {X 444.3606, Y 50.0328, Z -5.5000, A 0.000, B 0.000, C 0.000 }
gfCNCPoint4[3327] = {X 443.5314, Y 50.7763, Z -5.5000, A 0.000, B 0.000, C 0.000 }
gfCNCPoint4[3328] = {X 442.7495, Y 51.2994, Z -5.5000, A 0.000, B 0.000, C 0.000 }
gfCNCPoint4[3329] = {X 441.9067, Y 51.7174, Z -5.5000, A 0.000, B 0.000, C 0.000 }
gfCNCPoint4[3330] = {X 441.0171, Y 52.0232, Z -5.5000, A 0.000, B 0.000, C 0.000 }
gfCNCPoint4[3331] = {X 440.0673, Y 52.2155, Z -5.5000, A 0.000, B 0.000, C 0.000 }
gfCNCPoint4[3332] = {X 439.1005, Y 52.2800, Z -5.5000, A 0.000, B 0.000, C 0.000 }
gfCNCPoint4[3333] = {X 432.5144, Y 52.2800, Z -5.5000, A 0.000, B 0.000, C 0.000 }
gfCNCPoint4[3334] = {X 431.6034, Y 52.2228, Z -5.5000, A 0.000, B 0.000, C 0.000 }
gfCNCPoint4[3335] = {X 430.7067, Y 52.0520, Z -5.5000, A 0.000, B 0.000, C 0.000 }
gfCNCPoint4[3336] = {X 429.8384, Y 51.7703, Z -5.5000, A 0.000, B 0.000, C 0.000 }
gfCNCPoint4[3337] = {X 430.0168, Y 52.0769, Z -5.5000, A 0.000, B 0.000, C 0.000 }
gfCNCPoint4[3338] = {X 430.1862, Y 52.3887, Z -5.5000, A 0.000, B 0.000, C 0.000 }
gfCNCPoint4[3339] = {X 432.4638, Y 53.2762, Z -5.5000, A 0.000, B 0.000, C 0.000 }
gfCNCPoint4[3340] = {X 440.7638, Y 56.5693, Z -5.5000, A 0.000, B 0.000, C 0.000 }
gfCNCPoint4[3341] = {X 439.8787, Y 58.8002, Z -5.5000, A 0.000, B 0.000, C 0.000 }
gfCNCPoint4[3342] = {X 449.5094, Y 62.6213, Z -5.5000, A 0.000, B 0.000, C 0.000 }
gfCNCPoint4[3343] = {X 449.1113, Y 61.4464, Z -5.5000, A 0.000, B 0.000, C 0.000 }
gfCNCPoint4[3344] = {X 448.8668, Y 60.2304, Z -5.5000, A 0.000, B 0.000, C 0.000 }
gfCNCPoint4[3345] = {X 448.7798, Y 58.9930, Z -5.5000, A 0.000, B 0.000, C 0.000 }
gfCNCPoint4[3346] = {X 448.7796, Y 58.0000, Z -5.5000, A 0.000, B 0.000, C 0.000 }
gfCNCPoint4[3347] = {X 448.8564, Y 56.7833, Z -5.5000, A 0.000, B 0.000, C 0.000 }
gfCNCPoint4[3348] = {X 449.0855, Y 55.5859, Z -5.5000, A 0.000, B 0.000, C 0.000 }
gfCNCPoint4[3349] = {X 449.4632, Y 54.4268, Z -5.5000, A 0.000, B 0.000, C 0.000 }
gfCNCPoint4[3350] = {X 449.9837, Y 53.3244, Z -5.5000, A 0.000, B 0.000, C 0.000 }
gfCNCPoint4[3351] = {X 450.6386, Y 52.2961, Z -5.5000, A 0.000, B 0.000, C 0.000 }
gfCNCPoint4[3352] = {X 451.3887, Y 51.3890, Z -5.5000, A 0.000, B 0.000, C 0.000 }
gfCNCPoint4[3353] = {X 452.2434, Y 50.5796, Z -5.5000, A 0.000, B 0.000, C 0.000 }
gfCNCPoint4[3354] = {X 453.1901, Y 49.8800, Z -5.5000, A 0.000, B 0.000, C 0.000 }
gfCNCPoint4[3355] = {X 452.3731, Y 49.8442, Z -5.5000, A 0.000, B 0.000, C 0.000 }
gfCNCPoint4[3356] = {X 451.5735, Y 49.6724, Z -5.5000, A 0.000, B 0.000, C 0.000 }
gfCNCPoint4[3357] = {X 450.8138, Y 49.3696, Z -5.5000, A 0.000, B 0.000, C 0.000 }
gfCNCPoint4[3358] = {X 450.1154, Y 48.9441, Z -5.5000, A 0.000, B 0.000, C 0.000 }
gfCNCPoint4[3359] = {X 449.3503, Y 48.2496, Z -5.5000, A 0.000, B 0.000, C 0.000 }
gfCNCPoint4[3360] = {X 448.7486, Y 47.4095, Z -5.5000, A 0.000, B 0.000, C 0.000 }
gfCNCPoint4[3361] = {X 448.3373, Y 46.4616, Z -5.5000, A 0.000, B 0.000, C 0.000 }
gfCNCPoint4[3362] = {X 448.1732, Y 45.7588, Z -5.5000, A 0.000, B 0.000, C 0.000 }
gfCNCPoint4[3363] = {X 448.1146, Y 45.0395, Z -5.5000, A 0.000, B 0.000, C 0.000 }
gfCNCPoint4[3364] = {X 448.1149, Y 44.1416, Z -5.5000, A 0.000, B 0.000, C 0.000 }
gfCNCPoint4[3365] = {X 448.2252, Y 43.1751, Z -5.5000, A 0.000, B 0.000, C 0.000 }
gfCNCPoint4[3366] = {X 448.5250, Y 42.2496, Z -5.5000, A 0.000, B 0.000, C 0.000 }
gfCNCPoint4[3367] = {X 449.0024, Y 41.4020, Z -5.5000, A 0.000, B 0.000, C 0.000 }
gfCNCPoint4[3368] = {X 449.6384, Y 40.6660, Z -5.5000, A 0.000, B 0.000, C 0.000 }
gfCNCPoint4[3369] = {X 449.6384, Y 35.0338, Z -5.5000, A 0.000, B 0.000, C 0.000 }
gfCNCPoint4[3370] = {X 447.8169, Y 35.0338, Z -5.5000, A 0.000, B 0.000, C 0.000 }
gfCNCPoint4[3371] = {X 443.7929, Y 42.8687, Z -5.5000, A 0.000, B 0.000, C 0.000 }
gfCNCPoint4[3372] = {X 443.9303, Y 43.5107, Z -5.5000, A 0.000, B 0.000, C 0.000 }
gfCNCPoint4[3373] = {X 443.9803, Y 44.1653, Z -5.5000, A 0.000, B 0.000, C 0.000 }
gfCNCPoint4[3374] = {X 443.9805, Y 45.0000, Z -5.5000, A 0.000, B 0.000, C 0.000 }
gfCNCPoint4[3375] = {X 443.9242, Y 45.7387, Z -5.5000, A 0.000, B 0.000, C 0.000 }
gfCNCPoint4[3376] = {X 443.7568, Y 46.4603, Z -5.5000, A 0.000, B 0.000, C 0.000 }
gfCNCPoint4[3377] = {X 443.3474, Y 47.4038, Z -5.5000, A 0.000, B 0.000, C 0.000 }
gfCNCPoint4[3378] = {X 442.7493, Y 48.2405, Z -5.5000, A 0.000, B 0.000, C 0.000 }
gfCNCPoint4[3379] = {X 441.9891, Y 48.9332, Z -5.5000, A 0.000, B 0.000, C 0.000 }
gfCNCPoint4[3380] = {X 441.1006, Y 49.4513, Z -5.5000, A 0.000, B 0.000, C 0.000 }
gfCNCPoint4[3381] = {X 440.1232, Y 49.7716, Z -5.5000, A 0.000, B 0.000, C 0.000 }
gfCNCPoint4[3382] = {X 439.1005, Y 49.8800, Z -5.5000, A 0.000, B 0.000, C 0.000 }
gfCNCPoint4[3383] = {X 432.5144, Y 49.8800, Z -5.5000, A 0.000, B 0.000, C 0.000 }
gfCNCPoint4[3384] = {X 431.6014, Y 49.7938, Z -5.5000, A 0.000, B 0.000, C 0.000 }
gfCNCPoint4[3385] = {X 430.7206, Y 49.5383, Z -5.5000, A 0.000, B 0.000, C 0.000 }
gfCNCPoint4[3386] = {X 429.8343, Y 49.0782, Z -5.5000, A 0.000, B 0.000, C 0.000 }
gfCNCPoint4[3387] = {X 429.0603, Y 48.4473, Z -5.5000, A 0.000, B 0.000, C 0.000 }
gfCNCPoint4[3388] = {X 428.4309, Y 47.6720, Z -5.5000, A 0.000, B 0.000, C 0.000 }
gfCNCPoint4[3389] = {X 427.9725, Y 46.7848, Z -5.5000, A 0.000, B 0.000, C 0.000 }
gfCNCPoint4[3390] = {X 427.7197, Y 45.9083, Z -5.5000, A 0.000, B 0.000, C 0.000 }
gfCNCPoint4[3391] = {X 427.6344, Y 45.0000, Z -5.5000, A 0.000, B 0.000, C 0.000 }
gfCNCPoint4[3392] = {X 427.6344, Y 44.2089, Z -5.5000, A 0.000, B 0.000, C 0.000 }
gfCNCPoint4[3393] = {X 427.7263, Y 43.2661, Z -5.5000, A 0.000, B 0.000, C 0.000 }
gfCNCPoint4[3394] = {X 427.9987, Y 42.3588, Z -5.5000, A 0.000, B 0.000, C 0.000 }
gfCNCPoint4[3395] = {X 428.4412, Y 41.5212, Z -5.5000, A 0.000, B 0.000, C 0.000 }
gfCNCPoint4[3396] = {X 429.0371, Y 40.7849, Z -5.5000, A 0.000, B 0.000, C 0.000 }
gfCNCPoint4[3397] = {X 429.7641, Y 40.1776, Z -5.5000, A 0.000, B 0.000, C 0.000 }
gfCNCPoint4[3398] = {X 430.5947, Y 39.7222, Z -5.5000, A 0.000, B 0.000, C 0.000 }
gfCNCPoint4[3399] = {X 434.2536, Y 32.5605, Z -5.5000, A 0.000, B 0.000, C 0.000 }
gfCNCPoint4[3400] = {X 433.0335, Y 31.6542, Z -5.5000, A 0.000, B 0.000, C 0.000 }
gfCNCPoint4[3401] = {X 431.9384, Y 30.6003, Z -5.5000, A 0.000, B 0.000, C 0.000 }
gfCNCPoint4[3402] = {X 430.9860, Y 29.4160, Z -5.5000, A 0.000, B 0.000, C 0.000 }
gfCNCPoint4[3403] = {X 430.1916, Y 28.1203, Z -5.5000, A 0.000, B 0.000, C 0.000 }
gfCNCPoint4[3404] = {X 429.5682, Y 26.7343, Z -5.5000, A 0.000, B 0.000, C 0.000 }
gfCNCPoint4[3405] = {X 429.1257, Y 25.2803, Z -5.5000, A 0.000, B 0.000, C 0.000 }
gfCNCPoint4[3406] = {X 428.8014, Y 23.5412, Z -5.5000, A 0.000, B 0.000, C 0.000 }
gfCNCPoint4[3407] = {X 428.6564, Y 21.7780, Z -5.5000, A 0.000, B 0.000, C 0.000 }
gfCNCPoint4[3408] = {X 428.6923, Y 20.0093, Z -5.5000, A 0.000, B 0.000, C 0.000 }
gfCNCPoint4[3409] = {X 428.9088, Y 18.2534, Z -5.5000, A 0.000, B 0.000, C 0.000 }
gfCNCPoint4[3410] = {X 429.3035, Y 16.5289, Z -5.5000, A 0.000, B 0.000, C 0.000 }
gfCNCPoint4[3411] = {X 429.8217, Y 15.0579, Z -5.5000, A 0.000, B 0.000, C 0.000 }
gfCNCPoint4[3412] = {X 430.5206, Y 13.6636, Z -5.5000, A 0.000, B 0.000, C 0.000 }
gfCNCPoint4[3413] = {X 431.3891, Y 12.3681, Z -5.5000, A 0.000, B 0.000, C 0.000 }
gfCNCPoint4[3414] = {X 432.4135, Y 11.1921, Z -5.5000, A 0.000, B 0.000, C 0.000 }
gfCNCPoint4[3415] = {X 433.5451, Y 10.1796, Z -5.5000, A 0.000, B 0.000, C 0.000 }
gfCNCPoint4[3416] = {X 434.7921, Y 9.3131, Z -5.5000, A 0.000, B 0.000, C 0.000 }
gfCNCPoint4[3417] = {X 436.1357, Y 8.6057, Z -5.5000, A 0.000, B 0.000, C 0.000 }
gfCNCPoint4[3418] = {X 437.5557, Y 8.0679, Z -5.5000, A 0.000, B 0.000, C 0.000 }
gfCNCPoint4[3419] = {X 439.0309, Y 7.7079, Z -5.5000, A 0.000, B 0.000, C 0.000 }
gfCNCPoint4[3420] = {X 441.1775, Y 7.4109, Z -5.5000, A 0.000, B 0.000, C 0.000 }
gfCNCPoint4[3421] = {X 443.3425, Y 7.3143, Z -5.5000, A 0.000, B 0.000, C 0.000 }
gfCNCPoint4[3422] = {X 459.4468, Y 7.3102, Z -5.5000, A 0.000, B 0.000, C 0.000 }
gfCNCPoint4[3423] = {X 460.4096, Y 7.4063, Z -5.5000, A 0.000, B 0.000, C 0.000 }
gfCNCPoint4[3424] = {X 461.3345, Y 7.6909, Z -5.5000, A 0.000, B 0.000, C 0.000 }
gfCNCPoint4[3425] = {X 462.1848, Y 8.1526, Z -5.5000, A 0.000, B 0.000, C 0.000 }
gfCNCPoint4[3426] = {X 462.9272, Y 8.7733, Z -5.5000, A 0.000, B 0.000, C 0.000 }
gfCNCPoint4[3427] = {X 463.5322, Y 9.5285, Z -5.5000, A 0.000, B 0.000, C 0.000 }
gfCNCPoint4[3428] = {X 463.9759, Y 10.3884, Z -5.5000, A 0.000, B 0.000, C 0.000 }
gfCNCPoint4[3429] = {X 464.2317, Y 11.2687, Z -5.5000, A 0.000, B 0.000, C 0.000 }
gfCNCPoint4[3430] = {X 464.3179, Y 12.1814, Z -5.5000, A 0.000, B 0.000, C 0.000 }
gfCNCPoint4[3431] = {X 464.3179, Y 12.9780, Z -5.5000, A 0.000, B 0.000, C 0.000 }
gfCNCPoint4[3432] = {X 464.2174, Y 13.9635, Z -5.5000, A 0.000, B 0.000, C 0.000 }
gfCNCPoint4[3433] = {X 463.9199, Y 14.9085, Z -5.5000, A 0.000, B 0.000, C 0.000 }
gfCNCPoint4[3434] = {X 463.4376, Y 15.7739, Z -5.5000, A 0.000, B 0.000, C 0.000 }
gfCNCPoint4[3435] = {X 462.7906, Y 16.5240, Z -5.5000, A 0.000, B 0.000, C 0.000 }
gfCNCPoint4[3436] = {X 462.7903, Y 16.7697, Z -5.5000, A 0.000, B 0.000, C 0.000 }
gfCNCPoint4[3437] = {X 462.7907, Y 25.8813, Z -5.5000, A 0.000, B 0.000, C 0.000 }
gfCNCPoint4[3438] = {X 467.5907, Y 25.8811, Z -5.5000, A 0.000, B 0.000, C 0.000 }
gfCNCPoint4[3439] = {X 467.5913, Y 38.9910, Z -5.5000, A 0.000, B 0.000, C 0.000 }
gfCNCPoint4[3440] = {X 467.6015, Y 39.0069, Z -5.5000, A 0.000, B 0.000, C 0.000 }
gfCNCPoint4[3441] = {X 468.3506, Y 37.9855, Z -5.5000, A 0.000, B 0.000, C 0.000 }
gfCNCPoint4[3442] = {X 469.2267, Y 37.0706, Z -5.5000, A 0.000, B 0.000, C 0.000 }
gfCNCPoint4[3443] = {X 470.2148, Y 36.2780, Z -5.5000, A 0.000, B 0.000, C 0.000 }
gfCNCPoint4[3444] = {X 471.5271, Y 33.7093, Z -5.5000, A 0.000, B 0.000, C 0.000 }
gfCNCPoint4[3445] = {X 470.4797, Y 32.4130, Z -5.5000, A 0.000, B 0.000, C 0.000 }
gfCNCPoint4[3446] = {X 469.5658, Y 31.0194, Z -5.5000, A 0.000, B 0.000, C 0.000 }
gfCNCPoint4[3447] = {X 468.7943, Y 29.5422, Z -5.5000, A 0.000, B 0.000, C 0.000 }
gfCNCPoint4[3448] = {X 468.1729, Y 27.9958, Z -5.5000, A 0.000, B 0.000, C 0.000 }
gfCNCPoint4[3449] = {X 467.7076, Y 26.3956, Z -5.5000, A 0.000, B 0.000, C 0.000 }
gfCNCPoint4[3450] = {X 467.6476, Y 26.1387, Z -5.5000, A 0.000, B 0.000, C 0.000 }
gfCNCPoint4[3451] = {X 467.5907, Y 25.8811, Z -5.5000, A 0.000, B 0.000, C 0.000 }
gfCNCPoint4[3452] = {X 465.1907, Y 25.8812, Z -5.5000, A 0.000, B 0.000, C 0.000 }
gfCNCPoint4[3453] = {X 465.1913, Y 39.7482, Z -5.5000, A 0.000, B 0.000, C 0.000 }
gfCNCPoint4[3454] = {X 465.3907, Y 40.0179, Z -5.5000, A 0.000, B 0.000, C 0.000 }
gfCNCPoint4[3455] = {X 465.5774, Y 40.2966, Z -5.5000, A 0.000, B 0.000, C 0.000 }
gfCNCPoint4[3456] = {X 466.0634, Y 41.1919, Z -5.5000, A 0.000, B 0.000, C 0.000 }
gfCNCPoint4[3457] = {X 466.4196, Y 42.1462, Z -5.5000, A 0.000, B 0.000, C 0.000 }
gfCNCPoint4[3458] = {X 466.6392, Y 43.1408, Z -5.5000, A 0.000, B 0.000, C 0.000 }
gfCNCPoint4[3459] = {X 466.7178, Y 44.1564, Z -5.5000, A 0.000, B 0.000, C 0.000 }
gfCNCPoint4[3460] = {X 466.7179, Y 45.0000, Z -5.5000, A 0.000, B 0.000, C 0.000 }
gfCNCPoint4[3461] = {X 466.7033, Y 45.4609, Z -5.5000, A 0.000, B 0.000, C 0.000 }
gfCNCPoint4[3462] = {X 466.6596, Y 45.9200, Z -5.5000, A 0.000, B 0.000, C 0.000 }
gfCNCPoint4[3463] = {X 468.5433, Y 45.9200, Z -5.5000, A 0.000, B 0.000, C 0.000 }
gfCNCPoint4[3464] = {X 468.4996, Y 45.4609, Z -5.5000, A 0.000, B 0.000, C 0.000 }
gfCNCPoint4[3465] = {X 468.4850, Y 45.0000, Z -5.5000, A 0.000, B 0.000, C 0.000 }
gfCNCPoint4[3466] = {X 468.4850, Y 44.2089, Z -5.5000, A 0.000, B 0.000, C 0.000 }
gfCNCPoint4[3467] = {X 468.5580, Y 43.1798, Z -5.5000, A 0.000, B 0.000, C 0.000 }
gfCNCPoint4[3468] = {X 468.7759, Y 42.1714, Z -5.5000, A 0.000, B 0.000, C 0.000 }
gfCNCPoint4[3469] = {X 469.1341, Y 41.2038, Z -5.5000, A 0.000, B 0.000, C 0.000 }
gfCNCPoint4[3470] = {X 469.6255, Y 40.2966, Z -5.5000, A 0.000, B 0.000, C 0.000 }
gfCNCPoint4[3471] = {X 470.3102, Y 39.3876, Z -5.5000, A 0.000, B 0.000, C 0.000 }
gfCNCPoint4[3472] = {X 471.1282, Y 38.5964, Z -5.5000, A 0.000, B 0.000, C 0.000 }
gfCNCPoint4[3473] = {X 472.0595, Y 37.9424, Z -5.5000, A 0.000, B 0.000, C 0.000 }
gfCNCPoint4[3474] = {X 474.4565, Y 33.2506, Z -5.5000, A 0.000, B 0.000, C 0.000 }
gfCNCPoint4[3475] = {X 473.2245, Y 32.0060, Z -5.5000, A 0.000, B 0.000, C 0.000 }
gfCNCPoint4[3476] = {X 472.1526, Y 30.6211, Z -5.5000, A 0.000, B 0.000, C 0.000 }
gfCNCPoint4[3477] = {X 471.2565, Y 29.1165, Z -5.5000, A 0.000, B 0.000, C 0.000 }
gfCNCPoint4[3478] = {X 470.5495, Y 27.5143, Z -5.5000, A 0.000, B 0.000, C 0.000 }
gfCNCPoint4[3479] = {X 470.0420, Y 25.8382, Z -5.5000, A 0.000, B 0.000, C 0.000 }
gfCNCPoint4[3480] = {X 469.9882, Y 25.6081, Z -5.5000, A 0.000, B 0.000, C 0.000 }
gfCNCPoint4[3481] = {X 469.9372, Y 25.3774, Z -5.5000, A 0.000, B 0.000, C 0.000 }
gfCNCPoint4[3482] = {X 469.6262, Y 23.4829, Z -5.5000, A 0.000, B 0.000, C 0.000 }
gfCNCPoint4[3483] = {X 469.5012, Y 21.5671, Z -5.5000, A 0.000, B 0.000, C 0.000 }
gfCNCPoint4[3484] = {X 469.5634, Y 19.6483, Z -5.5000, A 0.000, B 0.000, C 0.000 }
gfCNCPoint4[3485] = {X 469.8121, Y 17.7447, Z -5.5000, A 0.000, B 0.000, C 0.000 }
gfCNCPoint4[3486] = {X 470.2450, Y 15.8743, Z -5.5000, A 0.000, B 0.000, C 0.000 }
gfCNCPoint4[3487] = {X 470.6914, Y 14.5430, Z -5.5000, A 0.000, B 0.000, C 0.000 }
gfCNCPoint4[3488] = {X 471.2621, Y 13.2600, Z -5.5000, A 0.000, B 0.000, C 0.000 }
gfCNCPoint4[3489] = {X 469.1179, Y 12.1817, Z -5.5000, A 0.000, B 0.000, C 0.000 }
gfCNCPoint4[3490] = {X 469.1885, Y 12.0430, Z -5.5000, A 0.000, B 0.000, C 0.000 }
gfCNCPoint4[3491] = {X 469.2603, Y 11.9049, Z -5.5000, A 0.000, B 0.000, C 0.000 }
gfCNCPoint4[3492] = {X 469.1140, Y 11.9049, Z -5.5000, A 0.000, B 0.000, C 0.000 }
gfCNCPoint4[3493] = {X 469.1170, Y 12.0433, Z -5.5000, A 0.000, B 0.000, C 0.000 }
gfCNCPoint4[3494] = {X 469.1179, Y 12.1817, Z -5.5000, A 0.000, B 0.000, C 0.000 }
gfCNCPoint4[3495] = {X 471.2621, Y 13.2600, Z -5.5000, A 0.000, B 0.000, C 0.000 }
gfCNCPoint4[3496] = {X 471.3228, Y 13.1407, Z -5.5000, A 0.000, B 0.000, C 0.000 }
gfCNCPoint4[3497] = {X 471.3845, Y 13.0219, Z -5.5000, A 0.000, B 0.000, C 0.000 }
gfCNCPoint4[3498] = {X 472.1257, Y 11.7667, Z -5.5000, A 0.000, B 0.000, C 0.000 }
gfCNCPoint4[3499] = {X 472.9867, Y 10.5906, Z -5.5000, A 0.000, B 0.000, C 0.000 }
gfCNCPoint4[3500] = {X 473.9593, Y 9.5049, Z -5.5000, A 0.000, B 0.000, C 0.000 }
gfCNCPoint4[3501] = {X 466.2074, Y 9.5049, Z -5.5000, A 0.000, B 0.000, C 0.000 }
gfCNCPoint4[3502] = {X 466.5690, Y 10.7171, Z -5.5000, A 0.000, B 0.000, C 0.000 }
gfCNCPoint4[3503] = {X 466.7150, Y 11.9735, Z -5.5000, A 0.000, B 0.000, C 0.000 }
gfCNCPoint4[3504] = {X 466.7172, Y 12.0775, Z -5.5000, A 0.000, B 0.000, C 0.000 }
gfCNCPoint4[3505] = {X 466.7179, Y 12.1814, Z -5.5000, A 0.000, B 0.000, C 0.000 }
gfCNCPoint4[3506] = {X 466.7179, Y 12.9779, Z -5.5000, A 0.000, B 0.000, C 0.000 }
gfCNCPoint4[3507] = {X 466.6192, Y 14.1732, Z -5.5000, A 0.000, B 0.000, C 0.000 }
gfCNCPoint4[3508] = {X 466.3255, Y 15.3360, Z -5.5000, A 0.000, B 0.000, C 0.000 }
gfCNCPoint4[3509] = {X 465.8449, Y 16.4349, Z -5.5000, A 0.000, B 0.000, C 0.000 }
gfCNCPoint4[3510] = {X 465.1903, Y 17.4399, Z -5.5000, A 0.000, B 0.000, C 0.000 }
gfCNCPoint4[3511] = {X 465.1907, Y 25.8812, Z -5.5000, A 0.000, B 0.000, C 0.000 }
gfCNCPoint4[3512] = {X 462.7907, Y 25.8813, Z -5.5000, A 0.000, B 0.000, C 0.000 }
gfCNCPoint4[3513] = {X 462.7913, Y 40.6635, Z -5.5000, A 0.000, B 0.000, C 0.000 }
gfCNCPoint4[3514] = {X 463.4321, Y 41.4050, Z -5.5000, A 0.000, B 0.000, C 0.000 }
gfCNCPoint4[3515] = {X 463.9118, Y 42.2596, Z -5.5000, A 0.000, B 0.000, C 0.000 }
gfCNCPoint4[3516] = {X 464.2110, Y 43.1928, Z -5.5000, A 0.000, B 0.000, C 0.000 }
gfCNCPoint4[3517] = {X 464.3178, Y 44.1670, Z -5.5000, A 0.000, B 0.000, C 0.000 }
gfCNCPoint4[3518] = {X 464.3179, Y 45.0000, Z -5.5000, A 0.000, B 0.000, C 0.000 }
gfCNCPoint4[3519] = {X 464.3082, Y 45.3090, Z -5.5000, A 0.000, B 0.000, C 0.000 }
gfCNCPoint4[3520] = {X 464.2788, Y 45.6167, Z -5.5000, A 0.000, B 0.000, C 0.000 }
gfCNCPoint4[3521] = {X 464.0485, Y 46.5992, Z -5.5000, A 0.000, B 0.000, C 0.000 }
gfCNCPoint4[3522] = {X 463.6209, Y 47.5134, Z -5.5000, A 0.000, B 0.000, C 0.000 }
gfCNCPoint4[3523] = {X 463.0145, Y 48.3200, Z -5.5000, A 0.000, B 0.000, C 0.000 }
gfCNCPoint4[3524] = {X 462.6627, Y 47.9934, Z -5.5000, A 0.000, B 0.000, C 0.000 }
gfCNCPoint4[3525] = {X 461.9835, Y 48.5889, Z -5.5000, A 0.000, B 0.000, C 0.000 }
gfCNCPoint4[3526] = {X 461.1970, Y 49.0331, Z -5.5000, A 0.000, B 0.000, C 0.000 }
gfCNCPoint4[3527] = {X 460.3364, Y 49.3073, Z -5.5000, A 0.000, B 0.000, C 0.000 }
gfCNCPoint4[3528] = {X 459.4379, Y 49.4000, Z -5.5000, A 0.000, B 0.000, C 0.000 }
gfCNCPoint4[3529] = {X 452.9945, Y 49.4000, Z -5.5000, A 0.000, B 0.000, C 0.000 }
gfCNCPoint4[3530] = {X 452.0154, Y 49.2897, Z -5.5000, A 0.000, B 0.000, C 0.000 }
gfCNCPoint4[3531] = {X 451.0854, Y 48.9643, Z -5.5000, A 0.000, B 0.000, C 0.000 }
gfCNCPoint4[3532] = {X 450.2511, Y 48.4400, Z -5.5000, A 0.000, B 0.000, C 0.000 }
gfCNCPoint4[3533] = {X 449.5544, Y 47.7433, Z -5.5000, A 0.000, B 0.000, C 0.000 }
gfCNCPoint4[3534] = {X 449.0302, Y 46.9091, Z -5.5000, A 0.000, B 0.000, C 0.000 }
gfCNCPoint4[3535] = {X 448.7048, Y 45.9791, Z -5.5000, A 0.000, B 0.000, C 0.000 }
gfCNCPoint4[3536] = {X 448.5945, Y 45.0000, Z -5.5000, A 0.000, B 0.000, C 0.000 }
gfCNCPoint4[3537] = {X 448.5949, Y 44.1483, Z -5.5000, A 0.000, B 0.000, C 0.000 }
gfCNCPoint4[3538] = {X 448.7053, Y 43.2275, Z -5.5000, A 0.000, B 0.000, C 0.000 }
gfCNCPoint4[3539] = {X 449.0063, Y 42.3503, Z -5.5000, A 0.000, B 0.000, C 0.000 }
gfCNCPoint4[3540] = {X 449.4844, Y 41.5556, Z -5.5000, A 0.000, B 0.000, C 0.000 }
gfCNCPoint4[3541] = {X 450.1184, Y 40.8789, Z -5.5000, A 0.000, B 0.000, C 0.000 }
gfCNCPoint4[3542] = {X 450.1184, Y 34.5538, Z -5.5000, A 0.000, B 0.000, C 0.000 }
gfCNCPoint4[3543] = {X 447.5238, Y 34.5538, Z -5.5000, A 0.000, B 0.000, C 0.000 }
gfCNCPoint4[3544] = {X 443.2766, Y 42.8232, Z -5.5000, A 0.000, B 0.000, C 0.000 }
gfCNCPoint4[3545] = {X 443.4441, Y 43.5071, Z -5.5000, A 0.000, B 0.000, C 0.000 }
gfCNCPoint4[3546] = {X 443.5005, Y 44.2089, Z -5.5000, A 0.000, B 0.000, C 0.000 }
gfCNCPoint4[3547] = {X 443.5005, Y 45.0000, Z -5.5000, A 0.000, B 0.000, C 0.000 }
gfCNCPoint4[3548] = {X 443.3902, Y 45.9791, Z -5.5000, A 0.000, B 0.000, C 0.000 }
gfCNCPoint4[3549] = {X 443.0647, Y 46.9091, Z -5.5000, A 0.000, B 0.000, C 0.000 }
gfCNCPoint4[3550] = {X 442.5405, Y 47.7434, Z -5.5000, A 0.000, B 0.000, C 0.000 }
gfCNCPoint4[3551] = {X 441.8438, Y 48.4401, Z -5.5000, A 0.000, B 0.000, C 0.000 }
gfCNCPoint4[3552] = {X 441.0096, Y 48.9643, Z -5.5000, A 0.000, B 0.000, C 0.000 }
gfCNCPoint4[3553] = {X 440.0796, Y 49.2897, Z -5.5000, A 0.000, B 0.000, C 0.000 }
gfCNCPoint4[3554] = {X 439.1005, Y 49.4000, Z -5.5000, A 0.000, B 0.000, C 0.000 }
gfCNCPoint4[3555] = {X 432.5144, Y 49.4000, Z -5.5000, A 0.000, B 0.000, C 0.000 }
gfCNCPoint4[3556] = {X 431.5353, Y 49.2897, Z -5.5000, A 0.000, B 0.000, C 0.000 }
gfCNCPoint4[3557] = {X 430.6053, Y 48.9643, Z -5.5000, A 0.000, B 0.000, C 0.000 }
gfCNCPoint4[3558] = {X 429.7711, Y 48.4401, Z -5.5000, A 0.000, B 0.000, C 0.000 }
gfCNCPoint4[3559] = {X 429.0743, Y 47.7434, Z -5.5000, A 0.000, B 0.000, C 0.000 }
gfCNCPoint4[3560] = {X 428.5501, Y 46.9091, Z -5.5000, A 0.000, B 0.000, C 0.000 }
gfCNCPoint4[3561] = {X 428.2247, Y 45.9791, Z -5.5000, A 0.000, B 0.000, C 0.000 }
gfCNCPoint4[3562] = {X 428.1144, Y 45.0000, Z -5.5000, A 0.000, B 0.000, C 0.000 }
gfCNCPoint4[3563] = {X 428.1148, Y 44.1483, Z -5.5000, A 0.000, B 0.000, C 0.000 }
gfCNCPoint4[3564] = {X 428.2132, Y 43.2816, Z -5.5000, A 0.000, B 0.000, C 0.000 }
gfCNCPoint4[3565] = {X 428.4806, Y 42.4514, Z -5.5000, A 0.000, B 0.000, C 0.000 }
gfCNCPoint4[3566] = {X 428.9065, Y 41.6903, Z -5.5000, A 0.000, B 0.000, C 0.000 }
gfCNCPoint4[3567] = {X 429.4741, Y 41.0281, Z -5.5000, A 0.000, B 0.000, C 0.000 }
gfCNCPoint4[3568] = {X 430.1613, Y 40.4909, Z -5.5000, A 0.000, B 0.000, C 0.000 }
gfCNCPoint4[3569] = {X 430.9408, Y 40.0998, Z -5.5000, A 0.000, B 0.000, C 0.000 }
gfCNCPoint4[3570] = {X 434.8817, Y 32.3860, Z -5.5000, A 0.000, B 0.000, C 0.000 }
gfCNCPoint4[3571] = {X 433.6221, Y 31.5161, Z -5.5000, A 0.000, B 0.000, C 0.000 }
gfCNCPoint4[3572] = {X 432.4895, Y 30.4863, Z -5.5000, A 0.000, B 0.000, C 0.000 }
gfCNCPoint4[3573] = {X 431.5043, Y 29.3148, Z -5.5000, A 0.000, B 0.000, C 0.000 }
gfCNCPoint4[3574] = {X 430.6838, Y 28.0224, Z -5.5000, A 0.000, B 0.000, C 0.000 }
gfCNCPoint4[3575] = {X 430.0428, Y 26.6323, Z -5.5000, A 0.000, B 0.000, C 0.000 }
gfCNCPoint4[3576] = {X 429.5927, Y 25.1692, Z -5.5000, A 0.000, B 0.000, C 0.000 }
gfCNCPoint4[3577] = {X 429.2772, Y 23.4782, Z -5.5000, A 0.000, B 0.000, C 0.000 }
gfCNCPoint4[3578] = {X 429.1362, Y 21.7638, Z -5.5000, A 0.000, B 0.000, C 0.000 }
gfCNCPoint4[3579] = {X 429.1711, Y 20.0439, Z -5.5000, A 0.000, B 0.000, C 0.000 }
gfCNCPoint4[3580] = {X 429.3815, Y 18.3366, Z -5.5000, A 0.000, B 0.000, C 0.000 }
gfCNCPoint4[3581] = {X 429.7653, Y 16.6598, Z -5.5000, A 0.000, B 0.000, C 0.000 }
gfCNCPoint4[3582] = {X 430.3281, Y 15.0962, Z -5.5000, A 0.000, B 0.000, C 0.000 }
gfCNCPoint4[3583] = {X 431.1031, Y 13.6262, Z -5.5000, A 0.000, B 0.000, C 0.000 }
gfCNCPoint4[3584] = {X 432.0751, Y 12.2783, Z -5.5000, A 0.000, B 0.000, C 0.000 }
gfCNCPoint4[3585] = {X 433.2253, Y 11.0789, Z -5.5000, A 0.000, B 0.000, C 0.000 }
gfCNCPoint4[3586] = {X 434.5313, Y 10.0513, Z -5.5000, A 0.000, B 0.000, C 0.000 }
gfCNCPoint4[3587] = {X 435.9676, Y 9.2154, Z -5.5000, A 0.000, B 0.000, C 0.000 }
gfCNCPoint4[3588] = {X 437.5062, Y 8.5876, Z -5.5000, A 0.000, B 0.000, C 0.000 }
gfCNCPoint4[3589] = {X 439.1173, Y 8.1801, Z -5.5000, A 0.000, B 0.000, C 0.000 }
gfCNCPoint4[3590] = {X 441.2214, Y 7.8889, Z -5.5000, A 0.000, B 0.000, C 0.000 }
gfCNCPoint4[3591] = {X 443.3434, Y 7.7943, Z -5.5000, A 0.000, B 0.000, C 0.000 }
gfCNCPoint4[3592] = {X 444.0367, Y 7.7902, Z -5.5000, A 0.000, B 0.000, C 0.000 }
gfCNCPoint4[3593] = {X 459.4468, Y 7.7902, Z -5.5000, A 0.000, B 0.000, C 0.000 }
gfCNCPoint4[3594] = {X 460.4239, Y 7.9003, Z -5.5000, A 0.000, B 0.000, C 0.000 }
gfCNCPoint4[3595] = {X 461.3520, Y 8.2251, Z -5.5000, A 0.000, B 0.000, C 0.000 }
gfCNCPoint4[3596] = {X 462.1846, Y 8.7482, Z -5.5000, A 0.000, B 0.000, C 0.000 }
gfCNCPoint4[3597] = {X 462.8799, Y 9.4436, Z -5.5000, A 0.000, B 0.000, C 0.000 }
gfCNCPoint4[3598] = {X 463.4031, Y 10.2761, Z -5.5000, A 0.000, B 0.000, C 0.000 }
gfCNCPoint4[3599] = {X 463.7278, Y 11.2043, Z -5.5000, A 0.000, B 0.000, C 0.000 }
gfCNCPoint4[3600] = {X 463.8379, Y 12.1814, Z -5.5000, A 0.000, B 0.000, C 0.000 }
gfCNCPoint4[3601] = {X 463.8377, Y 13.0201, Z -5.5000, A 0.000, B 0.000, C 0.000 }
gfCNCPoint4[3602] = {X 463.7299, Y 13.9469, Z -5.5000, A 0.000, B 0.000, C 0.000 }
gfCNCPoint4[3603] = {X 463.4292, Y 14.8301, Z -5.5000, A 0.000, B 0.000, C 0.000 }
gfCNCPoint4[3604] = {X 462.9489, Y 15.6300, Z -5.5000, A 0.000, B 0.000, C 0.000 }
gfCNCPoint4[3605] = {X 462.3108, Y 16.3107, Z -5.5000, A 0.000, B 0.000, C 0.000 }
gfCNCPoint4[3606] = {X 462.3103, Y 16.7692, Z -5.5000, A 0.000, B 0.000, C 0.000 }
gfCNCPoint4[3607] = {X 462.3113, Y 40.8766, Z -5.5000, A 0.000, B 0.000, C 0.000 }
gfCNCPoint4[3608] = {X 462.9556, Y 41.5657, Z -5.5000, A 0.000, B 0.000, C 0.000 }
gfCNCPoint4[3609] = {X 463.4381, Y 42.3762, Z -5.5000, A 0.000, B 0.000, C 0.000 }
gfCNCPoint4[3610] = {X 463.7368, Y 43.2710, Z -5.5000, A 0.000, B 0.000, C 0.000 }
gfCNCPoint4[3611] = {X 463.8379, Y 44.2089, Z -5.5000, A 0.000, B 0.000, C 0.000 }
gfCNCPoint4[3612] = {X 463.8379, Y 45.0000, Z -5.5000, A 0.000, B 0.000, C 0.000 }
gfCNCPoint4[3613] = {X 463.7612, Y 45.8182, Z -5.5000, A 0.000, B 0.000, C 0.000 }
gfCNCPoint4[3614] = {X 463.5336, Y 46.6079, Z -5.5000, A 0.000, B 0.000, C 0.000 }
gfCNCPoint4[3615] = {X 463.1632, Y 47.3415, Z -5.5000, A 0.000, B 0.000, C 0.000 }
gfCNCPoint4[3616] = {X 462.6627, Y 47.9934, Z -5.5000, A 0.000, B 0.000, C 0.000 }
gfCNCPoint4[3617] = {X 463.0145, Y 48.3200, Z -5.5000, A 0.000, B 0.000, C 0.000 }
gfCNCPoint4[3618] = {X 472.1884, Y 48.3200, Z -5.5000, A 0.000, B 0.000, C 0.000 }
gfCNCPoint4[3619] = {X 471.5820, Y 47.5134, Z -5.5000, A 0.000, B 0.000, C 0.000 }
gfCNCPoint4[3620] = {X 471.1544, Y 46.5992, Z -5.5000, A 0.000, B 0.000, C 0.000 }
gfCNCPoint4[3621] = {X 470.9241, Y 45.6167, Z -5.5000, A 0.000, B 0.000, C 0.000 }
gfCNCPoint4[3622] = {X 470.8947, Y 45.3090, Z -5.5000, A 0.000, B 0.000, C 0.000 }
gfCNCPoint4[3623] = {X 470.8850, Y 45.0000, Z -5.5000, A 0.000, B 0.000, C 0.000 }
gfCNCPoint4[3624] = {X 470.8850, Y 44.2089, Z -5.5000, A 0.000, B 0.000, C 0.000 }
gfCNCPoint4[3625] = {X 470.9769, Y 43.2661, Z -5.5000, A 0.000, B 0.000, C 0.000 }
gfCNCPoint4[3626] = {X 471.2492, Y 42.3588, Z -5.5000, A 0.000, B 0.000, C 0.000 }
gfCNCPoint4[3627] = {X 471.6917, Y 41.5212, Z -5.5000, A 0.000, B 0.000, C 0.000 }
gfCNCPoint4[3628] = {X 472.2877, Y 40.7849, Z -5.5000, A 0.000, B 0.000, C 0.000 }
gfCNCPoint4[3629] = {X 473.0147, Y 40.1776, Z -5.5000, A 0.000, B 0.000, C 0.000 }
gfCNCPoint4[3630] = {X 473.8453, Y 39.7222, Z -5.5000, A 0.000, B 0.000, C 0.000 }
gfCNCPoint4[3631] = {X 477.5001, Y 32.5683, Z -5.5000, A 0.000, B 0.000, C 0.000 }
gfCNCPoint4[3632] = {X 476.2823, Y 31.6587, Z -5.5000, A 0.000, B 0.000, C 0.000 }
gfCNCPoint4[3633] = {X 475.1890, Y 30.6027, Z -5.5000, A 0.000, B 0.000, C 0.000 }
gfCNCPoint4[3634] = {X 474.2379, Y 29.4170, Z -5.5000, A 0.000, B 0.000, C 0.000 }
gfCNCPoint4[3635] = {X 473.4440, Y 28.1208, Z -5.5000, A 0.000, B 0.000, C 0.000 }
gfCNCPoint4[3636] = {X 472.8202, Y 26.7347, Z -5.5000, A 0.000, B 0.000, C 0.000 }
gfCNCPoint4[3637] = {X 472.3764, Y 25.2809, Z -5.5000, A 0.000, B 0.000, C 0.000 }
gfCNCPoint4[3638] = {X 472.0519, Y 23.5417, Z -5.5000, A 0.000, B 0.000, C 0.000 }
gfCNCPoint4[3639] = {X 471.9068, Y 21.7783, Z -5.5000, A 0.000, B 0.000, C 0.000 }
